				IF bMoveOnlyForwardAfterError THEN
					IF  (
						(ABS(LMOD(WheelAxisRef.NcToPlc.ActPos,360.0/nSlotsCount)) > (360.0/nSlotsCount*0.01)) AND
						(ABS(LMOD(WheelAxisRef.NcToPlc.ActPos,360.0/nSlotsCount)) < (360.0/nSlotsCount*0.99))  
						)
						AND NOT (LMOD(WheelAxisRef.NcToPlc.ActPos,360.0/nSlotsCount) = 0) 
					THEN                       
						 mcWheelMoveAbsolute.Position:=WheelAxisRef.NcToPlc.ActPos+360.0/nSlotsCount-LMOD(WheelAxisRef.NcToPlc.ActPos,360.0/nSlotsCount);
					ELSE
						mcWheelMoveAbsolute.Position:=WheelAxisRef.NcToPlc.ActPos;				
					END_IF 
				ELSE
					IF lrLastKnownPosition<>0 AND (ABS(ABS(lrLastKnownPosition)-ABS(WheelAxisRef.NcToPlc.ActPos))<(360.0/nSlotsCount*3)) THEN
						mcWheelMoveAbsolute.Position:=lrLastKnownPosition;
						mcWheelMoveAbsolute.Velocity:=lrVelocity;
						mcWheelMoveAbsolute.Acceleration:=lrAcceleration;
						mcWheelMoveAbsolute.Deceleration:=lrDeceleration;
						mcWheelPower.Override:=20;
						
						nTestW1:=nTestW1+1;
						(*Jak jest w ponad połowie ruchu to przesuwa się do przodu*) //Być może będzie trzeba przesuwać rejestr
						IF WheelAxisRef.NcToPlc.ActPos-lrLastKnownPosition > ((360.0/nSlotsCount)/2) THEN
							mcWheelMoveAbsolute.Position	:=	lrLastKnownPosition + 360.0/nSlotsCount;
							bMoveForward 					:=	TRUE; //Informacja że przesuneło się w prawo
							nTestW2 := nTestW2 + 1;
						END_IF
						
					ELSE
						IF LMOD(WheelAxisRef.NcToPlc.ActPos,360.0/nSlotsCount)>(360.0/nSlotsCount/2) THEN
							mcWheelMoveAbsolute.Position:=WheelAxisRef.NcToPlc.ActPos+360.0/nSlotsCount-LMOD(WheelAxisRef.NcToPlc.ActPos,360.0/nSlotsCount);
							nTestW3 := nTestW3 + 1;
						ELSE
							mcWheelMoveAbsolute.Position:=WheelAxisRef.NcToPlc.ActPos-LMOD(WheelAxisRef.NcToPlc.ActPos,360.0/nSlotsCount);
							nTestW4 := nTestW4 + 1;
						END_IF
						mcWheelMoveAbsolute.Velocity:=lrVelocity;
						mcWheelMoveAbsolute.Acceleration:=lrAcceleration;
						mcWheelMoveAbsolute.Deceleration:=lrDeceleration;
						mcWheelPower.Override:=20;
					END_IF
				END_IF*)
END_ACTION

END_FUNCTION_BLOCK

// ---- POUs/FB/F_StringToWstringPL.TcPOU
FUNCTION F_StringToWstringPL : WSTRING
VAR_INPUT
	sInput	: STRING;
END_VAR
VAR
	iNum			: INT;	
//	iChar			: INT;
	iLen			: INT;
END_VAR

iLen	:=LEN(sInput);	//ilość znaków w stringu
FOR iNum:=0 TO iLen-1 DO
	CASE sInput[iNum] OF
		
		140://Ś
			F_StringToWstringPL[iNum]	:= 90+256;
		143://Ź
			F_StringToWstringPL[iNum]	:= 121+256;	
		156://ś
			F_StringToWstringPL[iNum]	:= 91+256;
		159://ź
			F_StringToWstringPL[iNum]	:= 122+256;
		163://Ł
			F_StringToWstringPL[iNum]	:= 65+256;
		165://Ą
			F_StringToWstringPL[iNum]	:= 4+256;
		175://Ż
			F_StringToWstringPL[iNum]	:= 123+256;
		179://ł
			F_StringToWstringPL[iNum]	:= 66+256;
		185://ą
			F_StringToWstringPL[iNum]	:= 5+256;
		191://ż
			F_StringToWstringPL[iNum]	:= 124+256;
		198://Ć
			F_StringToWstringPL[iNum]	:= 6+256;
		202://Ę
			F_StringToWstringPL[iNum]	:= 24+256;	
		209://Ń
			F_StringToWstringPL[iNum]	:= 67+256;
//		211://Ó - bez zmiany
		230://ć
			F_StringToWstringPL[iNum]	:= 7+256;
		234://ę
			F_StringToWstringPL[iNum]	:= 25+256;
		241://ń
			F_StringToWstringPL[iNum]	:= 68+256;

//		243://ó - bez zmiany
		
		ELSE
			F_StringToWstringPL[iNum]	:= sInput[iNum];
	END_CASE

END_FOR
F_StringToWstringPL[iLen]:= 0;//Dodane 0 - koniec wstringa



//F_StringToWstringPL:="";

//FOR iNum:=1 TO LEN(sInput) DO
//	iChar	:= F_ToASC(MID(sInput,1,iNum));
//	CASE iChar OF
//		140:
//			F_StringToWstringPL	:= WCONCAT(F_StringToWstringPL,"Ś");
//		143:
//			F_StringToWstringPL	:= WCONCAT(F_StringToWstringPL,"Ź");
//		156:
//			F_StringToWstringPL	:= WCONCAT(F_StringToWstringPL,"ś");
//		159:
//			F_StringToWstringPL	:= WCONCAT(F_StringToWstringPL,"ź");
//		163:
//			F_StringToWstringPL	:= WCONCAT(F_StringToWstringPL,"Ł");
//		165:
//			F_StringToWstringPL	:= WCONCAT(F_StringToWstringPL,"Ą");
//		175:
//			F_StringToWstringPL	:= WCONCAT(F_StringToWstringPL,"Ż");	
//		179:
//			F_StringToWstringPL	:= WCONCAT(F_StringToWstringPL,"ł");
//		185:
//			F_StringToWstringPL	:= WCONCAT(F_StringToWstringPL,"ą");
//		191:
//			F_StringToWstringPL	:= WCONCAT(F_StringToWstringPL,"ż");
//		198:
//			F_StringToWstringPL	:= WCONCAT(F_StringToWstringPL,"Ć");
//		202:
//			F_StringToWstringPL	:= WCONCAT(F_StringToWstringPL,"Ę");		
//		209:
//			F_StringToWstringPL	:= WCONCAT(F_StringToWstringPL,"Ń");
//		211:
//			F_StringToWstringPL	:= WCONCAT(F_StringToWstringPL,"Ó");
//		230:
//			F_StringToWstringPL	:= WCONCAT(F_StringToWstringPL,"ć");
//		234:
//			F_StringToWstringPL	:= WCONCAT(F_StringToWstringPL,"ę");
//		241:
//			F_StringToWstringPL	:= WCONCAT(F_StringToWstringPL,"ń");
//		243:
//			F_StringToWstringPL	:= WCONCAT(F_StringToWstringPL,"ó");

		
//		ELSE
//			F_StringToWstringPL	:= WCONCAT(F_StringToWstringPL,TO_WSTRING(MID(sInput,1,iNum)));
			
//	END_CASE
//END_FOR

END_FUNCTION

// ---- POUs/P20_ExhaustFan.TcPOU
PROGRAM P20_ExhaustFan
VAR
	(*****************Wentylator wyciągaowy*******************)
	QbExhaustSystemEnable					AT %Q*	:BOOL;		
	IbExhaustSystemSwitchNormalMode			AT %I*	:BOOL;		
	IbExhaustSystemSwitchExMode				AT %I*	:BOOL;		
	IbExhaustSystemReady					AT %I*	:BOOL;		
	IbExhaustSystemAlarm					AT %I*	:BOOL;		
	IbExhaustSystemFlowOk					AT %I*	:BOOL;		
	IbExhaustSystemAlarmLevel1				AT %I*	:BOOL;		
			
	fbSensorAirFlow							: FB_SensorFlow;
	
END_VAR


QbExhaustSystemEnable := VIS.bExEnableShow OR bExEnable;

aSensors();

ExSensorWarning[1].sDescription:='Alarm poziomu 1 detekcja gazu 10%DGW';
IF (IbExhaustSystemAlarmLevel1 AND QbExhaustSystemEnable) AND NOT ExSensorWarning[1].bWarning THEN
	ExSensorWarning[1].bWarning		:=	TRUE;
ELSIF ( NOT IbExhaustSystemAlarmLevel1 )AND ExSensorWarning[1].bAcknowledge THEN
	ExSensorWarning[1].bWarning		:=	FALSE;
	ExSensorWarning[1].bAcknowledge	:=	FALSE;
	VIS.uliWarningAcknowledge.24 	:=	FALSE;
ELSIF ExSensorWarning[1].bAcknowledge THEN
	ExSensorWarning[1].bAcknowledge	:=	TRUE;
END_IF


ExhaustFanError;
IF ExhaustFanError.bReset THEN
	ExhaustFanError.bError				:= FALSE;
	ExhaustFanError.udiStationID		:= 0;
	ExhaustFanError.nErrorCode			:= 0;
	ExhaustFanError.bReset				:= FALSE;
	ExhaustFanError.sErrorString		:= '';
	ExhaustFanError.sErrorString2		:= '';	
END_IF
IF IbExhaustSystemAlarm AND QbExhaustSystemEnable AND NOT VIS.bErrorOccure THEN
	ExhaustFanError.bError				:= TRUE;
	ExhaustFanError.udiStationID		:= 75;
	ExhaustFanError.nErrorCode			:= 372;
	ExhaustFanError.bReset				:= FALSE;
	ExhaustFanError.sErrorString		:= 'System wentylacji Ex - błąd - sprawdź szafę R4 Ex';
	ExhaustFanError.sErrorString2		:= '';
ELSIF NOT QbExhaustSystemEnable THEN
	ExhaustFanError.bError				:= FALSE;
END_IF

ACTION aSensors:
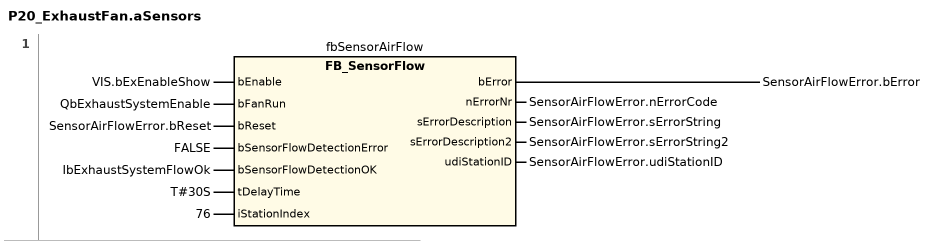
// NETWORK 1
fbSensorAirFlow(
    bEnable := VIS.bExEnableShow,
    bFanRun := QbExhaustSystemEnable,
    bReset := SensorAirFlowError.bReset,
    bSensorFlowDetectionError := FALSE,
    bSensorFlowDetectionOK := IbExhaustSystemFlowOk,
    tDelayTime := T#30S,
    iStationIndex := 76,
    nErrorNr => SensorAirFlowError.nErrorCode,
    sErrorDescription => SensorAirFlowError.sErrorString,
    sErrorDescription2 => SensorAirFlowError.sErrorString2,
    udiStationID => SensorAirFlowError.udiStationID); // FB_SensorFlow
SensorAirFlowError.bError := fbSensorAirFlow.bError;
END_ACTION

END_PROGRAM

// ---- POUs/FB/NewFBs/FB_SensorFlow.TcPOU
FUNCTION_BLOCK FB_SensorFlow
VAR_INPUT
	bEnable										:	BOOL;
	bFanRun										: 	BOOL;
	bReset										:	BOOL;
	bSensorFlowDetectionError				 	:	BOOL;			//Czujnik detekcji przeblywy bląd
	bSensorFlowDetectionOK					 	:	BOOL;			// Nie ma przeblywy
	tDelayTime									:	TIME;
	iStationIndex								:	UDINT;
END_VAR
	
VAR_OUTPUT
	bError										:	BOOL;
	nErrorNr									: 	UDINT;							//Nr błędu grzałki zasadniczej
	sErrorDescription							: 	STRING(200);	
	sErrorDescription2							: 	STRING(200);	
	udiStationID								:	UDINT;				// Nr stacji	
END_VAR
VAR
	tonSensorDelay								:	TON;
END_VAR

ACT_Cycle();
aStationID();

ACTION ACT_Cycle:
tonSensorDelay(IN:=(bEnable AND NOT bSensorFlowDetectionOK AND bFanRun),PT:=tDelayTime);

IF (NOT bError) THEN
	
	IF (bSensorFlowDetectionError) THEN
		bError 							:= FALSE;
		sErrorDescription 				:= 'Błąd czujnika przepływy';
		sErrorDescription2 				:= '';
		nErrorNr						:= 363;
	END_IF
	
	IF (tonSensorDelay.Q AND NOT bError) THEN
		bError 							:= FALSE;
		sErrorDescription 				:= 'Nie ma potwierdzenie przepływy od czujnika';
		sErrorDescription2 				:= '';
		nErrorNr						:= 364;
	END_IF
END_IF

IF (bReset) THEN
	bError 							:= FALSE;
	sErrorDescription 				:= '';
	sErrorDescription2 				:= '';
	nErrorNr						:= 0;
END_IF
END_ACTION

ACTION aStationID:
udiStationID	:=	iStationIndex;
END_ACTION

END_FUNCTION_BLOCK

// ---- POUs/P06_LidPuttedCheck.TcPOU
{attribute 'TcContextName' := 'PlcTask'}
PROGRAM P06_LidPuttedCheck
VAR
	fbLidPuttedCheck										: FB_VisionChecker;
	eLidPuttedCheckState									: E_Station; 			// Stan pracy podajnika platynek			
	eLidPuttedCheckRunningState								: E_CheckerState; 		// Stan pracy podajnika platynek
	fbLidPuttedCheckState									: FB_State;
	
	IbLidPuttedCheckHeightEncoderPulses 			AT %I*	: BOOL;	
	QbLidPuttedCheckHeightUpCmd 					AT %Q*	: BOOL; 				// Wyjście sterujące podnośnikiem sprawdzania platynki, Silnik w górę
	QbLidPuttedCheckHeightDownCmd 					AT %Q*	: BOOL; 				// Wyjście sterujące podnośnikiem sprawdzania platynki, Silnik w dół
	
	//Kamera do sprawdzania platynek
	IbLidPuttedCheckCameraError						AT %I*	: BOOL; 						
	IbLidPuttedCheckCameraGood						AT %I*	: BOOL; 						 
	IbLidPuttedCheckCameraBusy						AT %I*	: BOOL; 
	IuiLidPuttedCheckCameraProgram					AT %I*	: UINT; 
	
	QbLidPuttedCheckCameraTrigger					AT %Q*	: BOOL; 						
	QuiLidPuttedCheckCameraProgram					AT %Q*	: UINT; 
	QbLidPuttedCheckCameraChangeProgram				AT %Q*	: BOOL; 	
	
	TimerLidPuttedCheckEnable								: TOF;
	rtEnable												: R_TRIG;
	bTemp													: BOOL;

	IbLidPuttedCheck11Sensor						AT %I*	: BOOL; 	
	IbLidPuttedCheck12Sensor						AT %I*	: BOOL; 	
	IbLidPuttedCheck13Sensor						AT %I*	: BOOL; 	
	IbLidPuttedCheck21Sensor						AT %I*	: BOOL; 	
	IbLidPuttedCheck22Sensor						AT %I*	: BOOL; 	
	IbLidPuttedCheck23Sensor						AT %I*	: BOOL; 		
	
END_VAR

ACT_LidPuttedCheck();

(* BAZOWANIE - ZMIAN*)
rtEnable(CLK := fbLidPuttedCheck.bEnable, Q =>);
IF rtEnable.Q AND (P00_PackML.fbPMLAuto.ePMLState = Tc3_PackML.E_PMLState.ePMLState_IDLE OR 
   P00_PackML.fbPMLAuto.ePMLState = Tc3_PackML.E_PMLState.ePMLState_EXECUTE) THEN
   
   // VIS.bLidPuttedCheckHeightSet := TRUE;
	
ELSIF fbLidPuttedCheck.eState = E_Station.eHomingDone OR VIS.bErrorOccure THEN
	
   // VIS.bLidPuttedCheckHeightSet := FALSE;
	
END_IF
(*KONIEC BAZOWANIE - ZMIANA*)

(********* GENEROWANIE STANU STACJI DO WIZKI**********)
fbLidPuttedCheckState(
	eState					:= eLidPuttedCheckState , 
	bRun					:= P00_PackML.fbPMLAuto.ePMLState = Tc3_PackML.E_PMLState.ePMLState_EXECUTE,	
	eCheckerRunningState	:= eLidPuttedCheckRunningState , 
	sStateDesc				=> VIS.sLidPuttedCheckState,
	iState					=> VIS.iLidPuttedCheckState );
(***** KONIEC GENEROWANIE STANU STACJI DO WIZKI*******)	

(*Opoznienie wyłączanie enabla*)
TimerLidPuttedCheckEnable (IN := bLidPuttedCheckEnable , PT:=T#2S);

ACTION ACT_LidPuttedCheck:
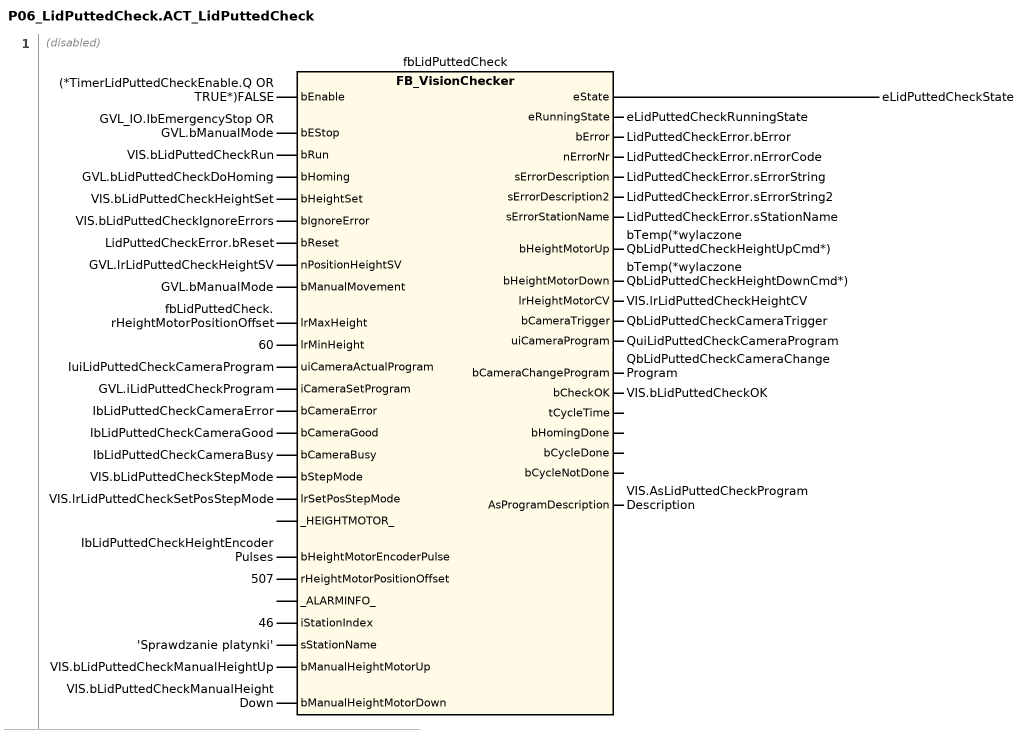
// NETWORK 1 (disabled)
// fbLidPuttedCheck(
//     bEnable := (*TimerLidPuttedCheckEnable.Q OR TRUE*)FALSE,
//     bEStop := GVL_IO.IbEmergencyStop OR GVL.bManualMode,
//     bRun := VIS.bLidPuttedCheckRun,
//     bHoming := GVL.bLidPuttedCheckDoHoming,
//     bHeightSet := VIS.bLidPuttedCheckHeightSet,
//     bIgnoreError := VIS.bLidPuttedCheckIgnoreErrors,
//     bReset := LidPuttedCheckError.bReset,
//     nPositionHeightSV := GVL.lrLidPuttedCheckHeightSV,
//     bManualMovement := GVL.bManualMode,
//     lrMaxHeight := fbLidPuttedCheck.rHeightMotorPositionOffset,
//     lrMinHeight := 60,
//     uiCameraActualProgram := IuiLidPuttedCheckCameraProgram,
//     iCameraSetProgram := GVL.iLidPuttedCheckProgram,
//     bCameraError := IbLidPuttedCheckCameraError,
//     bCameraGood := IbLidPuttedCheckCameraGood,
//     bCameraBusy := IbLidPuttedCheckCameraBusy,
//     bStepMode := VIS.bLidPuttedCheckStepMode,
//     lrSetPosStepMode := VIS.lrLidPuttedCheckSetPosStepMode,
//     bHeightMotorEncoderPulse := IbLidPuttedCheckHeightEncoderPulses,
//     rHeightMotorPositionOffset := 507,
//     iStationIndex := 46,
//     sStationName := 'Sprawdzanie platynki',
//     bManualHeightMotorUp := VIS.bLidPuttedCheckManualHeightUp,
//     bManualHeightMotorDown := VIS.bLidPuttedCheckManualHeightDown,
//     eRunningState => eLidPuttedCheckRunningState,
//     bError => LidPuttedCheckError.bError,
//     nErrorNr => LidPuttedCheckError.nErrorCode,
//     sErrorDescription => LidPuttedCheckError.sErrorString,
//     sErrorDescription2 => LidPuttedCheckError.sErrorString2,
//     sErrorStationName => LidPuttedCheckError.sStationName,
//     bHeightMotorUp => bTemp(*wylaczone QbLidPuttedCheckHeightUpCmd*),
//     bHeightMotorDown => bTemp(*wylaczone QbLidPuttedCheckHeightDownCmd*),
//     lrHeightMotorCV => VIS.lrLidPuttedCheckHeightCV,
//     bCameraTrigger => QbLidPuttedCheckCameraTrigger,
//     uiCameraProgram => QuiLidPuttedCheckCameraProgram,
//     bCameraChangeProgram => QbLidPuttedCheckCameraChangeProgram,
//     bCheckOK => VIS.bLidPuttedCheckOK,
//     AsProgramDescription => VIS.AsLidPuttedCheckProgramDescription); // FB_VisionChecker
// eLidPuttedCheckState := fbLidPuttedCheck.eState;
END_ACTION

END_PROGRAM

// ---- POUs/FB/FB_VisionChecker.TcPOU
(*
Nazwa:			FB_VisionChecker
Opis:			stacja sprawdzania platynek czujnikiem wizyjnym
Wersja:			v1.0
Data:			2023-05-30
Autor:			DP
Urzadzenia:		Czujnik wizyjny KEYENCE
Konfiguracja:	
Info:
- 
*)

FUNCTION_BLOCK FB_VisionChecker
VAR_INPUT
	bEnable:BOOL;				//Zezowlenie na pracę stacji sprawdzania
	bEStop:BOOL;				//Stop Awaryjny nieaktywny
	bRun:BOOL;					//Rozkaz łapania 	
	bHoming:BOOL;				//Zezwolenie na wykonanie bazowania i pozycjonowania stacji sprawdzania
	bHeightSet:BOOL;			//Ustaw wysokość
	bIgnoreError:BOOL;			//Ignorowania błędów cyklu pracy
	bReset:BOOL;				//Reset błędu, jeśli w stanie "eError"
	nPositionHeightSV:LREAL;	//Wysokość zadana na której ma znajdować się stacja sprawdzania
	bManualMovement:BOOL; 		//Uruchomienie trybu ruchów ręcznych
	lrMaxHeight:LREAL;			//Maksymalna wysokość stacji sprawdzania
	lrMinHeight:LREAL;			//Minimalna wysokość stacji sprawdzania
	uiCameraActualProgram:UINT;
	iCameraSetProgram:INT;
	bCameraError:BOOL; 
	bCameraGood:BOOL; 	
	bCameraBusy:BOOL; 	
	//StepMode
	bStepMode				: BOOL;		//Włączony tryb skokowy sterowania podnośnikami (tylko w serwisie)
	lrSetPosStepMode		: LREAL; 	//Ruch podnośnika o zadaną wartość w trybie krokowym (tylko w serwisie)
	
	_HEIGHTMOTOR_ :BOOL;	
	bHeightMotorEncoderPulse :BOOL;			//Sygnał impulsów enkodera siłownika
	rHeightMotorPositionOffset :REAL;		//Wysokość bazowani podnośnika

	_ALARMINFO_ :BOOL;
	iStationIndex:UDINT;					//Numer stacji 
	sStationName:STRING;					//Nazwa stacji	

END_VAR
VAR_OUTPUT	
	eState: E_Station;						//Stan ogólny bloku
	eRunningState: E_CheckerState;			//Stan stacji sprawdzania
	bError: BOOL;							//Błąd stacji
	nErrorNr: UDINT;						//Nr błędu stacji sprawdzania
	sErrorDescription:STRING(200);			//Opis błędu
	sErrorDescription2:STRING(200);			//Opis błędu
	sErrorStationName:STRING;				//Nazwa stacji
	bHeightMotorUp:BOOL;					//Sterowanie silnikiem podnośnika  - RUCH W GÓRĘ
	bHeightMotorDown:BOOL;					//Sterowanie silnikiem podnośnika  - RUCH W DÓŁ
	lrHeightMotorCV:LREAL;					//Aktualna wysokość stacji sprawdzania
	bCameraTrigger:BOOL; 
	uiCameraProgram:UINT; 
	bCameraChangeProgram:BOOL; 	
	bCheckOK:BOOL;							//Platynka OK
	tCycleTime:TIME;	
	bHomingDone:BOOL;						//Wymagane ponowne bazowanie (blad podczas bazowania lub stop awaryjny)
	bCycleDone:BOOL;
	bCycleNotDone:BOOL;
	AsProgramDescription: ARRAY [0..20] OF STRING;	// Opis programów

END_VAR
VAR
	tonHeightNoChange: TON; // Timer wykrycia braku ruchu siłownika zmiany wysokości stacji
	nLastPositionHeightCV: LREAL;// Pozycja podnośnika w poprzednim cyklu programu
	tonErrorHeightChange: TON; // Timer błędu podnośnika
	rtEncoderHomed:R_TRIG;
	tonCycleTimer:TON;
	rtrigCycleTimerRead:R_TRIG;
	tonTriggerDelay: TON;
	tonNotBusyDelay: TON;
	tonLidNOK: TON;
	tofMotorUpPermition: TOF;
	tofMotorDownPermition: TOF;
	tonLimitPosMinReachedDelay: TON;
	tonLimitPosMaxReachedDelay: TON;
	tonMaxHeight: TON;
	tonMinHeight: TON;
	
	//Podnośnik Jiesang	
	fbHeightMotorEncoder: FB_JiesangActuatorEncoder_1;	// Blok enkodera podnośnika chwytaka stabilizującego pod zakręcarką	
	bHeightMotorEncoderCounterReset:BOOL; 				// Sygnał resetu enkodera
	bHeightMotorEncoderHomed:BOOL;						// Informacja od enkodera że jest zbazowany

	eLastState: E_Station;								// Stan ogólny bloku
	eLastRunningState: E_CheckerState;					// Stan podbloku
	eLastStateTemp: E_Station;							// Stan ogólny bloku
	eLastRunningStateTemp: E_CheckerState;				// Stan podbloku	
	
	bStateError: BOOL;

	//Step Mode
	rtStepModeUp			: R_TRIG;
	rtStepModeDown			: R_TRIG;
	lrStepModeHeightMotorSV	: LREAL;
	bStepModeMoving			: BOOL;
	tofStepModeMoving		: TOF;	
	rtCheckingEnd			: R_TRIG;
	tonbCameraChangeProgram: TON;
	rtuiCameraActualProgram: R_TRIG;
	tonTryChangeProgram: TON;
	
	//Zmienne od EVENTLOGGER
	bAlarmInit 						: BOOL := TRUE; 
	nAlarmNumerator					: INT;
	arfbAlarm						: ARRAY[0..19] OF  FB_TcAlarm;		//Tablica bloczków błędów
	fbSourceInfo 					: FB_TcSourceInfo;
	iSourceInfo						: I_TcSourceInfo;
	sAlarmTest						: STRING;
	//Koniec zmiennych od EVENTLOGGER
END_VAR

VAR_IN_OUT
	bManualHeightMotorUp:BOOL;			//Ruch ręczny podnośnika stacji w górę
	bManualHeightMotorDown:BOOL;		//Ruch ręczny podnośnika stacji w dół
END_VAR

HeightMotor();
ErrorHandling();
Control();
Statistics();
Programs();

(*Zapisywanie ostatniego stanu*)
IF eLastStateTemp<>eState THEN
	eLastState := eLastStateTemp;
END_IF
eLastStateTemp := eState;
IF eLastRunningStateTemp<>eRunningState THEN
	eLastRunningState := eLastRunningStateTemp;
END_IF
eLastRunningStateTemp := eRunningState;
(*Koniec Zapisywanie ostatniego stanu*)

nLastPositionHeightCV:=lrHeightMotorCV;

ACTION Control:

	(** TIMERY**)
	rtEncoderHomed				(CLK:=bHeightMotorEncoderHomed,																Q=>);
	tonHeightNoChange			(IN:=((bHeightMotorUp OR bHeightMotorDown) AND (nLastPositionHeightCV=lrHeightMotorCV)), 	PT:=T#1S); 
	tonLimitPosMinReachedDelay	(IN:=(lrHeightMotorCV<=lrMinHeight) AND eState=E_Station.eHoming,							PT:=T#2S);
	tonLimitPosMaxReachedDelay	(IN:=(lrHeightMotorCV>=lrMaxHeight) AND eState=E_Station.eHoming,							PT:=T#2S);

	(*****Wyłączenie enable*****)
	IF NOT bEnable THEN
		IF eState <> E_Station.eDisabled AND eState <> E_Station.ePreparingToDisable THEN
				eState 							:=	E_Station.ePreparingToDisable; 
		END_IF	
	END_IF

	(*****Estop*****)
	IF NOT bEstop  THEN	
		IF eState <> E_Station.eAborted AND eState <> E_Station.eAborting AND eState <> E_Station.eDisabled THEN
				eState 							:=	E_Station.eAborting; 
		END_IF
	END_IF

	
	CASE eState OF
	/////////////////////////////	
		E_Station.eDisabled: 					// Stan nieaktywnosci (Stacja wyłączona) 
		
			IF bEnable THEN
				eState 							:=	E_Station.ePreparingToReady; 
			END_IF 
			
    /////////////////////////////	    
		E_Station.eAborted: 					// Stan bezpiecznego zatrzymania (po Abortingu) 

			IF bEStop THEN
				eState 							:=	E_Station.ePreparingToReady;
			END_IF
			
	/////////////////////////////	
		E_Station.eAborting:                 	// Stan bezpiecznego zatrzymywania (po EStopie)
			
			bHeightMotorUp						:=	FALSE;
			bHeightMotorDown					:=	FALSE;
			eState 								:=	E_Station.eAborted;  
			eRunningState						:=	E_CheckerState.eDisabled;
			
	/////////////////////////////			
		E_Station.eError:                 	 	// Stan błędu 	
	
			IF bReset THEN
				eState 							:=	E_Station.eResetting;
			ELSE
				ResetCommands();
			END_IF
			
	/////////////////////////////
		E_Station.eResetting:					// Stan resetowania bledu (po Errorze)
			
			bError := FALSE;
			IF NOT bError THEN
				nErrorNr 						:=	0;
   				sErrorDescription 				:=	'';
				eState 							:=	E_Station.ePreparingToReady;
			ELSE
				eState 							:=	E_Station.eError;
			END_IF
        
	/////////////////////////////
		E_Station.eManualMovement:     			// Stan ruchów manualnych  
       
			ManualMovements();
			//Wyjście z trybu serwisowego
			IF NOT bManualMovement THEN
				bHeightMotorUp					:=	FALSE;
				bHeightMotorDown				:=	FALSE;	
				eState							:=	E_Station.eReady;
			END_IF

	/////////////////////////////
		E_Station.eHoming:						// Stan bazowania 

			Homing();
			IF NOT bHoming AND NOT bHeightSet THEN
				bHeightMotorDown				:=	FALSE;
				bHeightMotorUp					:=	FALSE;
				eState							:=	E_Station.ePreparingToReady;
			END_IF		
			
	/////////////////////////////
		E_Station.eHomingDone:                  // Stan wykonania bazowania 
		
			bHeightMotorDown					:=	FALSE;
			bHeightMotorUp						:=	FALSE;
			bHeightMotorEncoderCounterReset		:=	FALSE;
			bHomingDone							:=	TRUE;
			IF NOT bHoming AND NOT bHeightSet THEN
			   eState							:=	E_Station.eReady;
			END_IF
			
	/////////////////////////////
		E_Station.ePreparingToReady:            // Stan przygotowywania do gotowosci (zawsze przed Ready)  
		
			eRunningState						:=	E_CheckerState.eReady;
			eState								:=	E_Station.eReady;	
			
	/////////////////////////////
		E_Station.ePreparingToDisable:          // Stan przygotowywania do nieaktywnosci (po wyłączeniu Enable) 
  
			bHeightMotorUp						:=	TRUE;
			bHeightMotorDown					:=	FALSE;	
			IF tonHeightNoChange.Q THEN
				bHeightMotorUp					:=	FALSE;
				eState							:=	E_Station.eDisabled;
				eRunningState					:=	E_CheckerState.eDisabled;
			END_IF	
				
	/////////////////////////////
		E_Station.eReady:						// Stan gotowosci 
			
			IF bRun AND NOT bCycleDone AND NOT bCycleNotDone THEN
				eState 							:=	E_Station.eStarting; 
			END_IF
			IF bHoming OR bHeightSet THEN
				eState 							:=	E_Station.eHoming; 
			END_IF
			IF bManualMovement THEN
				//Jeśli przejście w tryb ruchów manualnych przepisz wszystkie stany siłowników sterowanych przez moduł
				//aby zapobiec ewentualnym kolizjom po wejściu w tryb serwisowy
				bManualHeightMotorUp			:=	bHeightMotorUp;
				bManualHeightMotorDown			:=	bHeightMotorDown;
				eState 							:=	E_Station.eManualMovement; 
			END_IF
			IF NOT bRun THEN
				bCycleDone 						:=	FALSE;
				bCycleNotDone 					:=	FALSE;			
			END_IF
			
	/////////////////////////////
		E_Station.eStopping:					// Stan zatrzymywania 
			
			Running();
			bCameraTrigger						:= FALSE;
			bCheckOK							:= FALSE;
			eState								:=	E_Station.eReady;
			
	/////////////////////////////
		E_Station.eStarting:                  	// Stan uruchamiania (po Ready)
		
			eRunningState						:= E_CheckerState.eReady;
			eState								:= E_Station.eRunning; 

	/////////////////////////////
		E_Station.eRunning:               		// Stan wykonywania cyklu (po Startingu), w tym stanie osobny
 
			Running();
			IF NOT bRun THEN 					(*Przerywanie cyklu*)
				eState							:=	E_Station.eStopping;
				bCycleNotDone					:=	TRUE;
			END_IF
			(*IF bCycleDone OR bCycleNotDone THEN (*Cykl zakończony*)
				eState 				 := E_Station.eReady;
			END_IF*)						
			
	/////////////////////////////		
	END_CASE
END_ACTION

ACTION ErrorHandling:
// Alarm_0360	360	Error	Blokada podnośnika lub brak zasilania - sprawdź czujnik lub odblokuj mechanicznie
// Alarm_0361	361	Error	Wartość zadana wysokości jest większa od maksymalnej - zmień ustawienia w recepturze
// Alarm_0362	362	Error	Wartość zadana wysokości jest mniejsza od minimalnej - zmień ustawienia w recepturze

IF bAlarmInit THEN
    bAlarmInit := FALSE; 
	fbSourceInfo.Clear();
	fbSourceInfo.sName:=sStationName;//'Machine';
	fbSourceInfo.nId:=iStationIndex;//2700;
	// Alarm_0360	360	Error	Blokada podnośnika lub brak zasilania - sprawdź czujnik lub odblokuj mechanicznie
    arfbAlarm[0].CreateEx(stEventEntry := TC_EVENTS.AlarmClass.Alarm_0360, bWithConfirmation:= FALSE,  ipSourceInfo:= fbSourceInfo); 
	// Alarm_0361	361	Error	Wartość zadana wysokości jest większa od maksymalnej - zmień ustawienia w recepturze
	arfbAlarm[1].CreateEx(stEventEntry := TC_EVENTS.AlarmClass.Alarm_0361, bWithConfirmation:= FALSE,  ipSourceInfo:= fbSourceInfo);
	// Alarm_0362	362	Error	Wartość zadana wysokości jest mniejsza od minimalnej - zmień ustawienia w recepturze
	arfbAlarm[2].CreateEx(stEventEntry := TC_EVENTS.AlarmClass.Alarm_0362, bWithConfirmation:= FALSE,  ipSourceInfo:= fbSourceInfo);
END_IF

//OBSŁUGA BŁĘDÓW STACJI SPRAWDZANIA

//************LISTA BŁĘDÓW***************
bStateError:= (eState=E_Station.eError) OR (eState=E_Station.eResetting) OR bIgnoreError;

IF bEnable THEN
	// Alarm_0360	360	Error	Blokada podnośnika lub brak zasilania - sprawdź czujnik lub odblokuj mechanicznie
	//Error 1 - podnośnik nie porusza się pomimo wysterowania 
	tonErrorHeightChange(IN:=(bHeightMotorUp OR bHeightMotorDown) AND nLastPositionHeightCV=lrHeightMotorCV, PT:=T#3S);
	IF tonErrorHeightChange.Q THEN
		IF NOT arfbAlarm[0].bActive THEN
			bHeightMotorUp:=FALSE;
			bHeightMotorDown:=FALSE;
			arfbAlarm[0].Raise(nTimeStamp:=0);
		END_IF
	ELSE	
		IF  arfbAlarm[0].bActive AND bReset THEN
			arfbAlarm[0].Clear(nTimeStamp:=0, bResetConfirmation:= FALSE);
		END_IF	
// 		bHeightMotorUp:=FALSE;
// 		bHeightMotorDown:=FALSE;
// 		bError := TRUE;
// 		nErrorNr:=241;
// 		//nErrorNr := nErrorNr+iStationIndex;
// 		sErrorDescription:='Blokada podnośnika lub brak zasilania - sprawdź czujnik lub odblokuj mechanicznie';	
	END_IF
	// Alarm_0361	361	Error	Wartość zadana wysokości jest większa od maksymalnej - zmień ustawienia w recepturze
	//Error 7 - Bład nastaw max
	tonMaxHeight(IN:=nPositionHeightSV>lrMaxHeight AND NOT bHomingDone AND eState=E_Station.eStarting,PT:=T#0S);
	IF tonMaxHeight.Q THEN
		arfbAlarm[1].ipArguments.Clear() .AddLReal(lrMaxHeight);
		IF NOT arfbAlarm[1].bActive THEN
			bHeightMotorUp:=FALSE;
			bHeightMotorDown:=FALSE;
			arfbAlarm[1].Raise(nTimeStamp:=0);
		END_IF
	ELSE	
		IF  arfbAlarm[1].bActive AND bReset THEN
			arfbAlarm[1].Clear(nTimeStamp:=0, bResetConfirmation:= FALSE);
		END_IF	
// 		bHeightMotorUp:=FALSE;
// 		bHeightMotorDown:=FALSE;
// 		bError := TRUE;
// 		nErrorNr:=242;
// 		//nErrorNr := nErrorNr+iStationIndex;
// 		sErrorDescription:='Wartość zadana wysokości jest większa od maksymalnej - zmień ustawienia w recepturze';
// 		sErrorDescription2:=REAL_TO_STRING(LREAL_TO_INT(lrMaxHeight));
	END_IF
	// Alarm_0362	362	Error	Wartość zadana wysokości jest mniejsza od minimalnej - zmień ustawienia w recepturze
	//Error 8 - Bład nastaw min
	//tonMinHeight(IN:=nPositionHeightSV<lrMinHeight AND NOT bHomingDone AND eState=E_Station.eStarting,PT:=T#0S);
	//IF tonMinHeight.Q AND NOT bStateError THEN
	//	bHeightMotorUp:=FALSE;
	//	bHeightMotorDown:=FALSE;
	//	bError := TRUE;
	//	nErrorNr:=243;
	//	//nErrorNr := nErrorNr+iStationIndex;
	//	sErrorDescription:='Wartość zadana wysokości jest mniejsza od minimalnej - zmień ustawienia w recepturze';
	//	sErrorDescription2:=REAL_TO_STRING(LREAL_TO_INT(lrMinHeight));	
	//END_IF

ELSE
	bError := FALSE;
END_IF

	
//******************PRZEJŚCIE DO eERROR*****************************

IF bError AND NOT bStateError THEN
	IF eLastState = eRunning THEN
		bCycleNotDone := TRUE;
	END_IF
	eState := E_Station.eError;
END_IF

//****************WYŚWIETLANIE STATUSU BLEDU***********************

(*Wyświetlanie błedu na wyjściu*)
bError							:= FALSE;
FOR nAlarmNumerator := 0 TO 19 DO
	bError						:= bError OR arfbAlarm[nAlarmNumerator].bActive;
END_FOR

(*Przepisywanie nazwy stacji*)
sErrorStationName := sStationName;

//Jezeli nie zbazowane to potrzebne bazowanie
IF NOT bHeightMotorEncoderHomed  THEN
	bHomingDone:=FALSE;
END_IF
END_ACTION

ACTION HeightMotor:
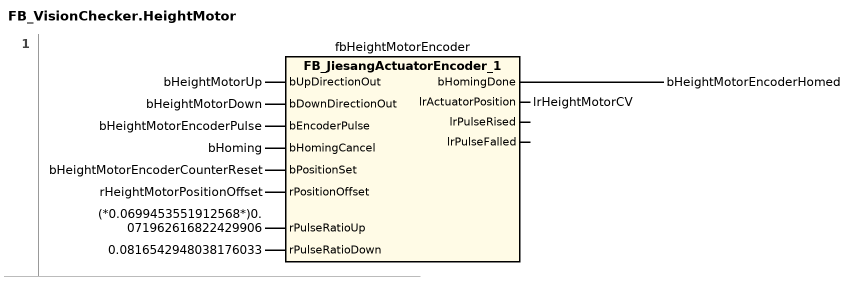
// NETWORK 1
fbHeightMotorEncoder(
    bUpDirectionOut := bHeightMotorUp,
    bDownDirectionOut := bHeightMotorDown,
    bEncoderPulse := bHeightMotorEncoderPulse,
    bHomingCancel := bHoming,
    bPositionSet := bHeightMotorEncoderCounterReset,
    rPositionOffset := rHeightMotorPositionOffset,
    rPulseRatioUp := (*0.0699453551912568*)0.071962616822429906,
    rPulseRatioDown := 0.0816542948038176033,
    lrActuatorPosition => lrHeightMotorCV); // FB_JiesangActuatorEncoder_1
bHeightMotorEncoderHomed := fbHeightMotorEncoder.bHomingDone;
END_ACTION

ACTION Homing:
//BAZOWANIE

	
//Podnoszenie stacji do maksymalnej pozycji
IF NOT bHeightMotorEncoderHomed OR rtEncoderHomed.Q THEN
	bHeightMotorUp:=TRUE;
	bHeightMotorDown:=FALSE;
	IF tonHeightNoChange.Q THEN
		bHeightMotorEncoderCounterReset:=TRUE;
		bHeightMotorUp:=FALSE;
    END_IF
	//Jesli enkoder zbazowany zakończ bazowanie	
	IF rtEncoderHomed.Q THEN
		bHeightMotorUp:=FALSE;
		bHeightMotorDown:=FALSE;
		eState:=E_Station.eHomingDone;
	END_IF		
		
//Po podniesieniu stacji opuszczanie do ustalonej wysokości
ELSIF bHeightMotorEncoderHomed THEN
	bHeightMotorEncoderCounterReset:=FALSE;
	bHeightMotorUp:=lrHeightMotorCV<=nPositionHeightSV;
	bHeightMotorDown:=lrHeightMotorCV>=nPositionHeightSV;
	//Kiedy stacja osiągnie wysokość zadaną
	IF ABS(lrHeightMotorCV-nPositionHeightSV)<1 OR tonLimitPosMaxReachedDelay.Q OR tonLimitPosMinReachedDelay.Q THEN
		bHeightMotorDown:=FALSE;
		bHeightMotorUp:=FALSE;
		eState:=E_Station.eHomingDone;
	END_IF			
END_IF
END_ACTION

ACTION ManualMovements:

//W trybie ruchów manualnych wykonuj ruchy za pomocą rozkazów manualnych
IF NOT bRun THEN
	eRunningState		:=	E_CheckerState.eReady;
	bCameraTrigger		:=	FALSE;
	bCheckOK			:=	FALSE;
	bHeightMotorUp		:=	bManualHeightMotorUp;
	bHeightMotorDown	:=	bManualHeightMotorDown;
ELSE	//Kasuje zeby po cyklu nic sie nie poruszało
	bManualHeightMotorUp  := FALSE;
	bManualHeightMotorDown  := FALSE;
END_IF


IF bHoming OR bHeightSet THEN
	eState:=E_Station.eHoming;
END_IF
	
Running();
ManualMovementsStepMode();
	
//Zabezpieczenie przed kolizją stacji poprzez ruch podnośnika	
IF bHeightMotorDown AND lrHeightMotorCV<=lrMinHeight AND NOT bHoming AND NOT bHeightSet THEN
	bHeightMotorDown:=FALSE;
END_IF	

IF bHeightMotorUp AND lrHeightMotorCV>=lrMaxHeight AND NOT bHoming AND NOT bHeightSet THEN
	bHeightMotorUp:=FALSE;
END_IF
END_ACTION

ACTION ManualMovementsStepMode:
bManualHeightMotorUp;
bManualHeightMotorDown;
bStepMode;		
lrSetPosStepMode;

// Limity
IF lrSetPosStepMode < 1			THEN	lrSetPosStepMode := 1;	END_IF
IF lrSetPosStepMode > 10		THEN	lrSetPosStepMode := 10;	END_IF

// Zabezpieczenie przed zbyt szybkim włączaniem
tofStepModeMoving				(IN := bStepModeMoving,					PT:=T#500MS);

// Możliwe włączenie jeżeli zakończyło poprzedni ruch
rtStepModeUp					(CLK :=	bStepMode AND NOT tofStepModeMoving.Q	AND bManualHeightMotorUp,	Q=>);
rtStepModeDown					(CLK :=	bStepMode AND NOT tofStepModeMoving.Q 	AND bManualHeightMotorDown,	Q=>);

// Włączenie ruchu w górę
IF rtStepModeUp.Q THEN
	bStepModeMoving				:= TRUE;
	bManualHeightMotorUp		:= FALSE;
	bManualHeightMotorDown		:= FALSE;
	lrStepModeHeightMotorSV		:= lrHeightMotorCV	+	lrSetPosStepMode;
END_IF

// Włączenie ruchu w dół
IF rtStepModeDown.Q THEN
	bStepModeMoving				:= TRUE;
	bManualHeightMotorUp		:= FALSE;
	bManualHeightMotorDown		:= FALSE;
	lrStepModeHeightMotorSV		:= lrHeightMotorCV	-	lrSetPosStepMode;
END_IF
// DODAĆ RESET bStepModeMoving PO BLEDZIE!
// Ruch w górę !SPRAWDZIC ZNAKI!
IF bStepModeMoving THEN
	bHeightMotorUp				:=	lrHeightMotorCV	<=	lrStepModeHeightMotorSV;
	bHeightMotorDown			:=	lrHeightMotorCV	>=	lrStepModeHeightMotorSV;	
	
	IF ABS(lrHeightMotorCV-lrStepModeHeightMotorSV) < 0.5	OR	// Pozycja osiągnięta (co do 1mm)
			(lrHeightMotorCV<=lrMinHeight)				OR 	// Pozycja poniżej minimalnej
			(lrHeightMotorCV>=lrMaxHeight) 					// Pozycja powyżej maksymalnej
	THEN
		bHeightMotorDown		:= FALSE;
		bHeightMotorUp			:= FALSE;
		bStepModeMoving			:= FALSE;
	END_IF	
END_IF
END_ACTION

ACTION Programs:
tonbCameraChangeProgram	(IN:=bCameraChangeProgram,PT:=T#1S);
tonTryChangeProgram	(IN:=uiCameraActualProgram <> uiCameraProgram AND NOT bCameraChangeProgram, PT:=T#5S);
rtuiCameraActualProgram	(CLK:=uiCameraActualProgram <> uiCameraProgram,	Q=>);
uiCameraProgram	:=	INT_TO_UINT(iCameraSetProgram);

IF rtuiCameraActualProgram.Q	 OR  tonTryChangeProgram.Q THEN
	bCameraChangeProgram	:=	TRUE;
END_IF
IF tonbCameraChangeProgram.Q THEN
	bCameraChangeProgram	:=	FALSE;
END_IF

(*Narzędzia*)
AsProgramDescription[0] := '1. opak:225082(elite), platynka:241081(~55mm)';
AsProgramDescription[1] := '2. opak:220505(wega), platynka:soraya 240964(54mm)';
AsProgramDescription[2] := '3. opak:220395(shine), platynka:bielenda 241181(57mm)';
AsProgramDescription[3] := '4. opak:rezerwa, platynka:rezerwa';
AsProgramDescription[4] := '5. opak:rezerwa, platynka:rezerwa';
AsProgramDescription[5] := '6. opak:rezerwa, platynka:rezerwa';
AsProgramDescription[6] := '7. opak:rezerwa, platynka:rezerwa';
AsProgramDescription[7] := '8. opak:rezerwa, platynka:rezerwa';
AsProgramDescription[8] := '9. opak:220601(200ml), platynka:240234(~ mm)';
AsProgramDescription[9] := '10. opak:220395(shine), platynka:soraya 240965(57mm)';
AsProgramDescription[10] := '11. opak:rezerwa, platynka:rezerwa';
AsProgramDescription[11] := '12. opak:rezerwa, platynka:rezerwa';
AsProgramDescription[12] := '13. opak:rezerwa, platynka:rezerwa';
AsProgramDescription[13] := '14. opak:rezerwa, platynka:rezerwa';
AsProgramDescription[14] := '15. opak:rezerwa, platynka:rezerwa';
END_ACTION

ACTION ResetCommands:

bStepModeMoving 			:= FALSE;
bHeightMotorDown			:= FALSE;
bHeightMotorUp				:= FALSE;
bManualHeightMotorUp		:= FALSE;
bManualHeightMotorDown		:= FALSE;
END_ACTION

ACTION Running:

//Timery
tofMotorUpPermition		(IN:=	bHeightMotorDown,								PT:=T#250MS);
tofMotorDownPermition	(IN:=	bHeightMotorUp,									PT:=T#250MS);
tonTriggerDelay			(IN:=	eRunningState=E_CheckerState.eFormPresent,		PT:=T#50MS);
tonNotBusyDelay			(IN:=	tonTriggerDelay.Q AND NOT bCameraBusy,
																				PT:=T#50MS);
tonLidNOK				(IN:=	eRunningState=E_CheckerState.eFormPresent,
																				PT:=T#50MS);				

CASE eRunningState OF
	
	E_CheckerState.eDisabled:
	
		eRunningState		:=	E_CheckerState.eReady;
	
	//SPRAWDZANIEGOTOWY DO PRACY
	E_CheckerState.eReady:
		
		IF bRun THEN
			eRunningState	:=	E_CheckerState.eFormPresent;	
		END_IF

	//WYKRYTO SLOIK
	E_CheckerState.eFormPresent:
	
		bCameraTrigger		:= TRUE;
		IF	tonTriggerDelay.Q THEN
			IF tonNotBusyDelay.Q AND bCameraGood THEN
				eRunningState	:=	E_CheckerState.eLidOK;		
			ELSIF tonNotBusyDelay.Q  THEN
				eRunningState	:=	E_CheckerState.eLidNOK;	
			END_IF	
		END_IF
		
	
	//BUTELKA W FORMATCE
	E_CheckerState.eBottleOK:
	;
	
	//PLATYNKA OK
	E_CheckerState.eLidOK:
	
		bCheckOK	:= TRUE;
		bCycleDone	:= TRUE;	
	
	//PLATYNKA NOK
	E_CheckerState.eLidNOK:

		bCheckOK	:= FALSE;	
		bCycleDone	:= TRUE;
		
	//NASADKA OK
	E_CheckerState.eCapOK:
	;
		
	//NASADKA NOK
	E_CheckerState.eCapNOK:
	;		

	E_CheckerState.eChecking:
	;
		
END_CASE
END_ACTION

ACTION Statistics:

rtrigCycleTimerRead(CLK:=eRunningState=E_CheckerState.eLidOK OR eRunningState=E_CheckerState.eLidNOK);
IF rtrigCycleTimerRead.Q THEN
		tCycleTime:=tonCycleTimer.ET;
END_IF
tonCycleTimer(IN:=eState>E_Station.eReady,PT:=T#1D);
END_ACTION

END_FUNCTION_BLOCK

// ---- POUs/P07_CapPusher.TcPOU
(*
Nazwa:			P07_CapPusher
Opis:			Wvijak nasadek z sorteram wibracyjnym
Wersja:			v0.1
Data:			2025-11-03
Autor:			DP
Urzadzenia:		
Konfiguracja:	
Info:
- 
*)
PROGRAM P07_CapPusher
VAR_INPUT
	//Szlaban
	//...
	
	//Podajnik
	//...
	
	//Zakrecanie
	//..

END_VAR
VAR
	(*****************SZLABAN*******************)
	fbCapPusherGate										: FB_SpringGateV2;
	QbCapPusherGate										AT %Q*: BOOL; 			// Wyjście sterujące 

	(*******************PODAJNIK*********************)
	fbCapPusherFeeder									: FB_CapPusherFeeder;
	fbCapPusherFeederState								: FB_State;	
	eCapPusherFeederState								: E_Station;
	eCapPusherFeederRunningState						: E_CapFeederState; 	// Stan pracy 
	QbCapPusherFeederSorterVibrator 					AT %Q*: BOOL; 			// Wyjście sterujące 
	QbCapPusherFeederSorterVibrator2 					AT %Q*: BOOL; 			// Wyjście sterujące 	
	QbCapPusherFeederSorterAir 							AT %Q*: BOOL; 			// Wyjście sterujące 
	IbCapPusherFeederHopperSensor						: BOOL; 					
	IbCapPusherFeederWheelSensor						: BOOL; 			
	IbCapPusherFeederSleeveSensor					: BOOL; 
	QnCapPusherFeederVelocitySV 						AT %Q*: UDINT; 			// Nastawa prędkości
	InCapPusherFeederVelocityCV 						AT %I*: UDINT;		
	InCapPusherFeederSTW 								AT %I*: UINT; 			// Statusword transportera wejściowo wyjściowego
	QnCapPusherFeederCTW 								AT %Q*: UINT;  			// Controlword transportera we/wy
	IbCapPusherFeederWcState							AT %I*: BOOL; 			// Statusword transportera wejściowo wyjściowego
	TimerCapPusherFeederEnable							: TOF;
	rtCapPusherFeederEnable								: R_TRIG;
	tonCapPusherFeederEnable							: TON;
	
	(*******ZAKRECANIE**********)
	fbCapPusher											: FB_CapPusher;
	fbCapPusherState									: FB_State;	
	eCapPusherState										: E_Station;
	eCapPusherRunningState								: E_GripperScrewer; 	// Stan pracy 	

	QbCapPusher											AT %Q*: BOOL; 	
	QbCapPusherBlockActuator							AT %Q*: BOOL; 	
	QbCapPusherFormPositioning							AT %Q*: BOOL; 	
	
	IbCapPusherFormSensor								: BOOL; 
	IbCapPusherCapSensor								: BOOL; 
	IbCapPusherUpSensor									: BOOL; 
	IbCapPusherDownSensor								: BOOL; 
	IbCapPusherBlockActuatorOnSensor					: BOOL; 
	IbCapPusherBlockActuatorOffSensor					: BOOL; 
	IbCapPusherFormPositioningUpSensor					: BOOL; 
	IbCapPusherFormPositioningDownSensor				: BOOL; 
	TimerCapPusherEnable								: TOF;
	rtCapPusherEnable									: R_TRIG;
	tonCapPusherEnable									: TON;
	
	(*RFID*)
	//Przed
	bReadedCard 										: BOOL;				
	nReadedCard											: ULINT;	
	fbReader   											: FB_IfmIoLinkRfid;
	AusiReaderInputData  								AT %I* : ARRAY[0..27] OF USINT;
	IbReaderTagPresent									AT %I* : BOOL;
	IBReaderErrorValue									AT %I* : BYTE;
	IbReaderCmdEnd										AT %I* : BOOL;
	IBReaderDataCounterIn								AT %I* : BYTE;
	IbReaderCmdStartAck									AT %I* : BOOL;
	IbReaderCmdStart									AT %Q* : BOOL;
	IBReaderCmmandValue									AT %Q* : BYTE;
	IBReaderDataCounterOut								AT %Q* : BYTE;
	AusiReaderOutputData  								AT %Q* : ARRAY[0..27] OF USINT;	

	(*Lampy*)
	QbCapPusherRedSignalizationLamp 					AT %Q* : BOOL;				
	QbCapPusherGreenSignalizationLamp 					AT %Q* : BOOL;					
	QbCapPusherYellowSignalizationLamp 					AT %Q* : BOOL;							
	
	(*Przyciski*)

	(*Safety*)
		

	QbCapPusherDoors0Close								AT %Q* :BOOL;		// Rozkaz zamkniecia 
	
	(*Zawór główny*)
	QbCapPusherCompressedAir							AT %Q*		:BOOL;		
	IbCapPusherCompressedAirOK 							AT %I*		:BOOL;		//Zasilanie powietrzem sprężonym OK	
	
	(*Zasilanie*)
	IbCapPusherFuseFB1OK								AT %I* :BOOL;		//		
	IbCapPusherFuseFB2OK								AT %I* :BOOL;		//	
	IbCapPusherFuseFB3OK								AT %I* :BOOL;		//	
	
	(*DI wyspy pneumatycznej*)
	QABPneumaticCapPusherEB1ValveCoils 						AT %Q* 	: ARRAY[1..5] OF BYTE;	
	IABPneumaticCapPusherEB1DigitalInput 					AT %I* 	: ARRAY[1..4] OF BYTE;
	IuiPneumaticCapPusherEB1State							AT %I* 	: UINT;	

	(*Czujniki formatek*)
	IbCapPusherThirdFormSensor	 							: BOOL; 		// Czujnik dojazdu 3 formatki
	
	(*Manual*)
	
	(****Inne***)

	
END_VAR

aPowerSupply();
aButtons();
aPneumatics();
aRFID();
aRFID_FB();
aSafety();
aSignalization();
aLimits();
a1_Gate();
a1_GateTime();
a2_Feeder();
a3_Capping();
aWarnings();

(*BAZOWANIE - ZMIAN*)
//SSzlaban
//...
//Podajnik
tonCapPusherFeederEnable (IN:=bCapPusherEnable,PT:=T#5S); 
rtCapPusherFeederEnable(CLK:=tonCapPusherFeederEnable.Q,Q=>);
IF rtCapPusherFeederEnable.Q AND (P00_PackML.fbPMLAuto.ePMLState = E_PMLState.ePMLState_IDLE OR P00_PackML.fbPMLAuto.ePMLState = E_PMLState.ePMLState_EXECUTE)   THEN
	VIS_CP.bCapPusherFeederHeightSet:=TRUE;
ELSIF fbCapPusherFeeder.eState=E_Station.eHomingDone	OR	VIS.bErrorOccure THEN
 	VIS_CP.bCapPusherFeederHeightSet:=FALSE;
END_IF
//Zakrecanie
tonCapPusherEnable (IN:=bCapPusherEnable,PT:=T#5S); 
rtCapPusherEnable(CLK:=tonCapPusherEnable.Q,Q=>);
IF rtCapPusherEnable.Q AND (P00_PackML.fbPMLAuto.ePMLState = E_PMLState.ePMLState_IDLE OR P00_PackML.fbPMLAuto.ePMLState = E_PMLState.ePMLState_EXECUTE)   THEN
	VIS_CP.bCapPusherHeightSet:=TRUE;
ELSIF fbCapPusher.eState=E_Station.eHomingDone	OR	VIS.bErrorOccure THEN
 	VIS_CP.bCapPusherHeightSet:=FALSE;
END_IF
(*KONIEC BAZOWANIE - ZMIANA*)

(*Opoznienie wyłączanie enabla*)
//Szlaban
//..
//Podajnik
TimerCapPusherFeederEnable	(IN:=bCapPusherEnable,	PT:=T#2S);
//Zakrecanie
TimerCapPusherEnable		(IN:=bCapPusherEnable, PT:=T#2S);

(*Staty*)
//Szlaban
//...
//Podajnik
fbCapPusherFeederState(
	eState							:=	eCapPusherFeederState , 
	bRun							:=	VIS_CP.bCapPusherFeederRun,	
	eCapFeederRunningState			:=	eCapPusherFeederRunningState , 
	sStateDesc						=>	VIS_CP.sCapPusherFeederState,
	iState							=>	VIS_CP.iCapPusherFeederState);	

//Zakrecanie
fbCapPusherState(
	eState							:=	eCapPusherState , 
	bRun							:=	VIS_CP.bCapPusherRun,	
	eGripperScrewerRunningState		:=	eCapPusherRunningState , 
	sStateDesc						=>	VIS_CP.sCapPusherState,
	iState							=>	VIS_CP.iCapPusherState);	


(********KASOWANIE ROZKAZÓW CYKLI*********)
//Szlaban
//...
//Podajnik
//...
//Zakrecanie
IF fbCapPusher.bCycleDone1 AND bManualMode THEN
	VIS_CP.bCapPusherRun 		:= FALSE;
END_IF

ACTION a1_Gate:
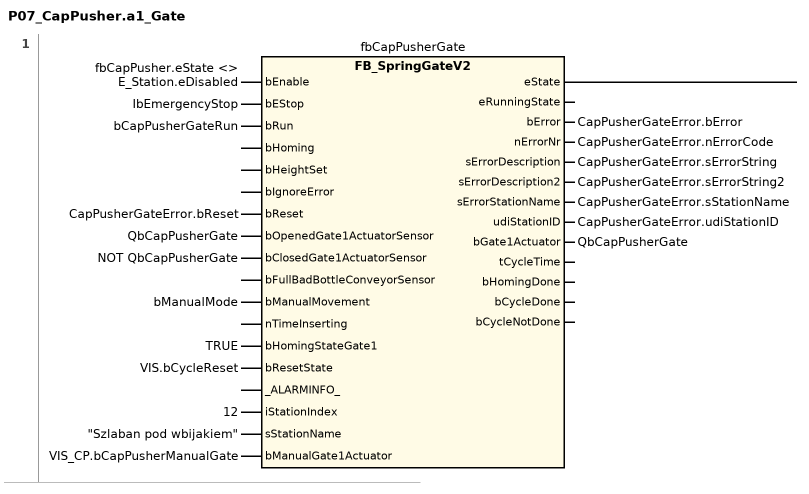
// NETWORK 1
fbCapPusherGate(
    bEnable := fbCapPusher.eState <> E_Station.eDisabled,
    bEStop := IbEmergencyStop,
    bRun := bCapPusherGateRun,
    bReset := CapPusherGateError.bReset,
    bOpenedGate1ActuatorSensor := QbCapPusherGate,
    bClosedGate1ActuatorSensor := NOT QbCapPusherGate,
    bManualMovement := bManualMode,
    bHomingStateGate1 := TRUE,
    bResetState := VIS.bCycleReset,
    iStationIndex := 12,
    sStationName := "Szlaban pod wbijakiem",
    bManualGate1Actuator := VIS_CP.bCapPusherManualGate,
    bError => CapPusherGateError.bError,
    nErrorNr => CapPusherGateError.nErrorCode,
    sErrorDescription => CapPusherGateError.sErrorString,
    sErrorDescription2 => CapPusherGateError.sErrorString2,
    sErrorStationName => CapPusherGateError.sStationName,
    udiStationID => CapPusherGateError.udiStationID,
    bGate1Actuator => QbCapPusherGate); // FB_SpringGateV2
END_ACTION

ACTION a1_GateTime:

fbCapPusherGate.nTimeInserting	:=	300;
END_ACTION

ACTION a2_Feeder:
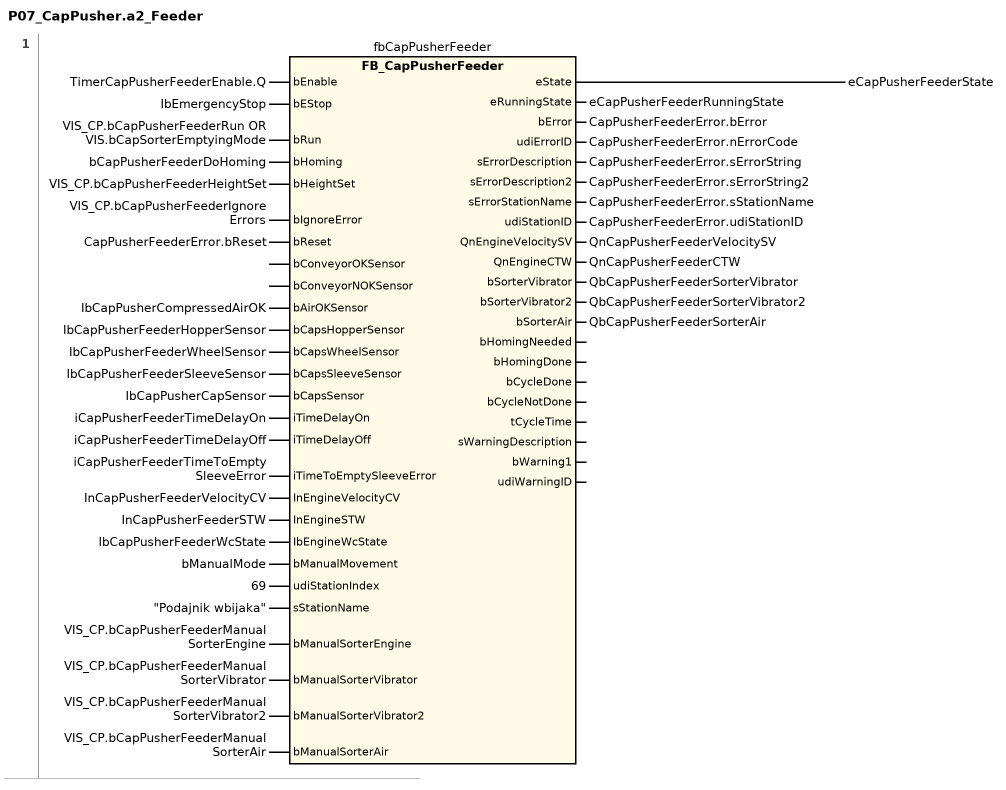
// NETWORK 1
fbCapPusherFeeder(
    bEnable := TimerCapPusherFeederEnable.Q,
    bEStop := IbEmergencyStop,
    bRun := VIS_CP.bCapPusherFeederRun OR VIS.bCapSorterEmptyingMode,
    bHoming := bCapPusherFeederDoHoming,
    bHeightSet := VIS_CP.bCapPusherFeederHeightSet,
    bIgnoreError := VIS_CP.bCapPusherFeederIgnoreErrors,
    bReset := CapPusherFeederError.bReset,
    bAirOKSensor := IbCapPusherCompressedAirOK,
    bCapsHopperSensor := IbCapPusherFeederHopperSensor,
    bCapsWheelSensor := IbCapPusherFeederWheelSensor,
    bCapsSleeveSensor := IbCapPusherFeederSleeveSensor,
    bCapsSensor := IbCapPusherCapSensor,
    iTimeDelayOn := iCapPusherFeederTimeDelayOn,
    iTimeDelayOff := iCapPusherFeederTimeDelayOff,
    iTimeToEmptySleeveError := iCapPusherFeederTimeToEmptySleeveError,
    InEngineVelocityCV := InCapPusherFeederVelocityCV,
    InEngineSTW := InCapPusherFeederSTW,
    IbEngineWcState := IbCapPusherFeederWcState,
    bManualMovement := bManualMode,
    udiStationIndex := 69,
    sStationName := "Podajnik wbijaka",
    bManualSorterEngine := VIS_CP.bCapPusherFeederManualSorterEngine,
    bManualSorterVibrator := VIS_CP.bCapPusherFeederManualSorterVibrator,
    bManualSorterVibrator2 := VIS_CP.bCapPusherFeederManualSorterVibrator2,
    bManualSorterAir := VIS_CP.bCapPusherFeederManualSorterAir,
    eRunningState => eCapPusherFeederRunningState,
    bError => CapPusherFeederError.bError,
    udiErrorID => CapPusherFeederError.nErrorCode,
    sErrorDescription => CapPusherFeederError.sErrorString,
    sErrorDescription2 => CapPusherFeederError.sErrorString2,
    sErrorStationName => CapPusherFeederError.sStationName,
    udiStationID => CapPusherFeederError.udiStationID,
    QnEngineVelocitySV => QnCapPusherFeederVelocitySV,
    QnEngineCTW => QnCapPusherFeederCTW,
    bSorterVibrator => QbCapPusherFeederSorterVibrator,
    bSorterVibrator2 => QbCapPusherFeederSorterVibrator2,
    bSorterAir => QbCapPusherFeederSorterAir); // FB_CapPusherFeeder
eCapPusherFeederState := fbCapPusherFeeder.eState;
END_ACTION

ACTION a3_Capping:
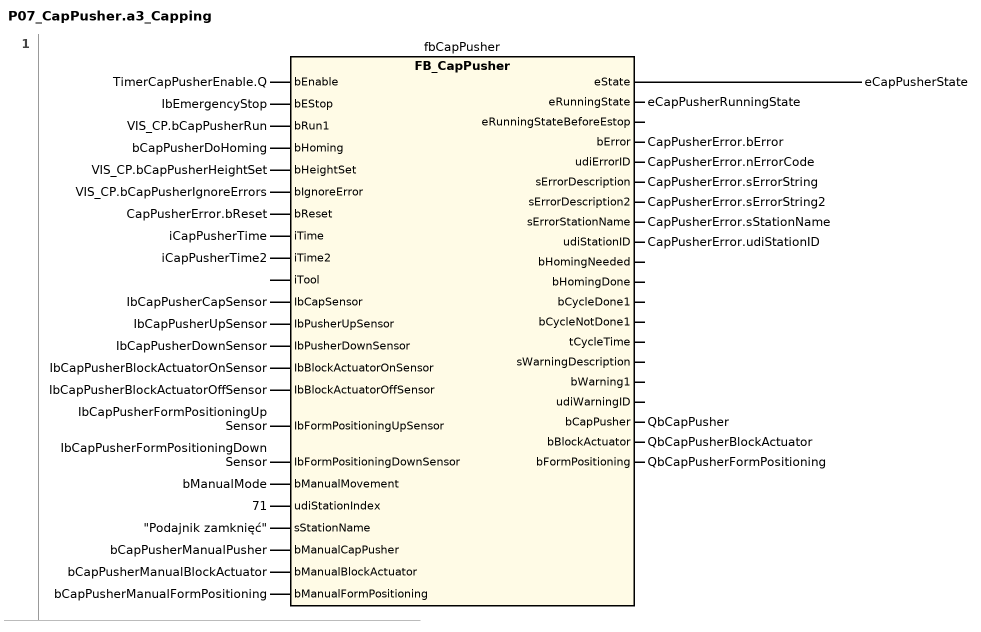
// NETWORK 1
fbCapPusher(
    bEnable := TimerCapPusherEnable.Q,
    bEStop := IbEmergencyStop,
    bRun1 := VIS_CP.bCapPusherRun,
    bHoming := bCapPusherDoHoming,
    bHeightSet := VIS_CP.bCapPusherHeightSet,
    bIgnoreError := VIS_CP.bCapPusherIgnoreErrors,
    bReset := CapPusherError.bReset,
    iTime := iCapPusherTime,
    iTime2 := iCapPusherTime2,
    IbCapSensor := IbCapPusherCapSensor,
    IbPusherUpSensor := IbCapPusherUpSensor,
    IbPusherDownSensor := IbCapPusherDownSensor,
    IbBlockActuatorOnSensor := IbCapPusherBlockActuatorOnSensor,
    IbBlockActuatorOffSensor := IbCapPusherBlockActuatorOffSensor,
    IbFormPositioningUpSensor := IbCapPusherFormPositioningUpSensor,
    IbFormPositioningDownSensor := IbCapPusherFormPositioningDownSensor,
    bManualMovement := bManualMode,
    udiStationIndex := 71,
    sStationName := "Podajnik zamknięć",
    bManualCapPusher := bCapPusherManualPusher,
    bManualBlockActuator := bCapPusherManualBlockActuator,
    bManualFormPositioning := bCapPusherManualFormPositioning,
    eRunningState => eCapPusherRunningState,
    bError => CapPusherError.bError,
    udiErrorID => CapPusherError.nErrorCode,
    sErrorDescription => CapPusherError.sErrorString,
    sErrorDescription2 => CapPusherError.sErrorString2,
    sErrorStationName => CapPusherError.sStationName,
    udiStationID => CapPusherError.udiStationID,
    bCapPusher => QbCapPusher,
    bBlockActuator => QbCapPusherBlockActuator,
    bFormPositioning => QbCapPusherFormPositioning); // FB_CapPusher
eCapPusherState := fbCapPusher.eState;
END_ACTION

ACTION aButtons:

END_ACTION

ACTION aLimits:
(*
Nazwa:			aLimits
Opis:			Zabezpieczenia
Wersja:			v1.0
Data:			2023-11-24
Autor:			DP
Urzadzenia:		
Zmiany:	

Info:
*)

(**** Limity i zabezpieczenia***)
END_ACTION

ACTION aPneumatics:
// Do podpięcia według kolejności
QbCapPusherGate;
QbCapPusherFeederSorterAir;
QbCapPusher;			
QbCapPusherBlockActuator;	
QbCapPusherFormPositioning;

(*************************** CapPusher EB1 **************************************)
// Wyspa 1 - dozowanie
IuiPneumaticCapPusherEB1State;
QABPneumaticCapPusherEB1ValveCoils[1].0	:= QbCapPusher;
QABPneumaticCapPusherEB1ValveCoils[1].1 := NOT QbCapPusher;
QABPneumaticCapPusherEB1ValveCoils[1].2 := QbCapPusherBlockActuator;
QABPneumaticCapPusherEB1ValveCoils[1].3 ;
QABPneumaticCapPusherEB1ValveCoils[1].4 := QbCapPusherFormPositioning;
QABPneumaticCapPusherEB1ValveCoils[1].5 ;
QABPneumaticCapPusherEB1ValveCoils[1].6 := NOT QbCapPusherGate;
QABPneumaticCapPusherEB1ValveCoils[1].7 := QbCapPusherGate; 
QABPneumaticCapPusherEB1ValveCoils[2].0 ;				
QABPneumaticCapPusherEB1ValveCoils[2].1 ;
QABPneumaticCapPusherEB1ValveCoils[2].2 ;
QABPneumaticCapPusherEB1ValveCoils[2].3 ;
QABPneumaticCapPusherEB1ValveCoils[2].4 ;											
QABPneumaticCapPusherEB1ValveCoils[2].5 ;
QABPneumaticCapPusherEB1ValveCoils[2].6 ;
QABPneumaticCapPusherEB1ValveCoils[2].7 ;
QABPneumaticCapPusherEB1ValveCoils[3].0 ;
QABPneumaticCapPusherEB1ValveCoils[3].1 ;
QABPneumaticCapPusherEB1ValveCoils[3].2 ;
QABPneumaticCapPusherEB1ValveCoils[3].3 ;
QABPneumaticCapPusherEB1ValveCoils[3].4 ; 
QABPneumaticCapPusherEB1ValveCoils[3].5 ;
QABPneumaticCapPusherEB1ValveCoils[3].6 ;
QABPneumaticCapPusherEB1ValveCoils[3].7 ;                                               
QABPneumaticCapPusherEB1ValveCoils[4].0	;		                                
QABPneumaticCapPusherEB1ValveCoils[4].1 ;                                       
QABPneumaticCapPusherEB1ValveCoils[4].2	;		                                
QABPneumaticCapPusherEB1ValveCoils[4].3 ;                                      
QABPneumaticCapPusherEB1ValveCoils[4].4 ;		                                
QABPneumaticCapPusherEB1ValveCoils[4].5 ;        
QABPneumaticCapPusherEB1ValveCoils[4].6 ;		
QABPneumaticCapPusherEB1ValveCoils[4].7 ; 
                                                              
(*********************Koniec CapPusher EB1 **************************************) 


//Zawór głównego powietrza
QbCapPusherCompressedAir	:=	IbEmergencyStop AND QbCapPusherFeederSorterAir;

(*************************** EB1 **************************************)
// Wyspa 1 - 52N8
IuiPneumaticCapPusherEB1State;
//DI1
IbCapPusherFeederHopperSensor		:=	IABPneumaticCapPusherEB1DigitalInput[1].0;	
IbCapPusherFeederWheelSensor		:=	NOT IABPneumaticCapPusherEB1DigitalInput[1].1;	
IbCapPusherFeederSleeveSensor		:=	IABPneumaticCapPusherEB1DigitalInput[1].2;	
										IABPneumaticCapPusherEB1DigitalInput[1].3;
IbCapPusherUpSensor					:=	IABPneumaticCapPusherEB1DigitalInput[1].4;	
IbCapPusherDownSensor				:=	IABPneumaticCapPusherEB1DigitalInput[1].5;	
IbCapPusherCapSensor				:=	IABPneumaticCapPusherEB1DigitalInput[1].6;	
										;IABPneumaticCapPusherEB1DigitalInput[1].7;	
//DI2                                           
IbCapPusherBlockActuatorOffSensor	:=	IABPneumaticCapPusherEB1DigitalInput[2].0;	
IbCapPusherBlockActuatorOnSensor	:=	IABPneumaticCapPusherEB1DigitalInput[2].1;	
IbCapPusherFormSensor				:=	IABPneumaticCapPusherEB1DigitalInput[2].2;	
IbCapPusherFormPositioningDownSensor:=	IABPneumaticCapPusherEB1DigitalInput[2].3;	
IbCapPusherFormPositioningUpSensor	:=	IABPneumaticCapPusherEB1DigitalInput[2].4;	
;	IABPneumaticCapPusherEB1DigitalInput[2].5;		
;	IABPneumaticCapPusherEB1DigitalInput[2].6;		
;	IABPneumaticCapPusherEB1DigitalInput[2].7;	

// Wyspa 1 - 52N8A
IuiPneumaticCapPusherEB1State;
//DI1
;	IABPneumaticCapPusherEB1DigitalInput[3].0;	
;	IABPneumaticCapPusherEB1DigitalInput[3].1;	
;	IABPneumaticCapPusherEB1DigitalInput[3].2;	
;	IABPneumaticCapPusherEB1DigitalInput[3].3;
;	IABPneumaticCapPusherEB1DigitalInput[3].4;	
;	IABPneumaticCapPusherEB1DigitalInput[3].5;		
;	IABPneumaticCapPusherEB1DigitalInput[3].6;		
;	IABPneumaticCapPusherEB1DigitalInput[3].7;
//DI2                                               		
;	IABPneumaticCapPusherEB1DigitalInput[4].0;
;	IABPneumaticCapPusherEB1DigitalInput[4].0;	
;	IABPneumaticCapPusherEB1DigitalInput[4].1;	
;	IABPneumaticCapPusherEB1DigitalInput[4].2;	
;	IABPneumaticCapPusherEB1DigitalInput[4].3;	
;	IABPneumaticCapPusherEB1DigitalInput[4].4;
;	IABPneumaticCapPusherEB1DigitalInput[4].5;		
;	IABPneumaticCapPusherEB1DigitalInput[4].6;		
	IABPneumaticCapPusherEB1DigitalInput[4].7;	
(*********************Koniec EB2 **************************************)
END_ACTION

ACTION aPowerSupply:


	//Dodane do głwnych
	IbCapPusherFuseFB1OK	; //Przekaznik kontroli faz
	IbCapPusherFuseFB2OK	; //Kontrola poprawności faz
	IbCapPusherFuseFB3OK	; //Blok bezpiecznikowy
END_ACTION

ACTION aRFID:
(*Przepisanie bity wykrycia karty*)
bReadedCard 		:= IbReaderTagPresent AND fbReader.bCodeReaded;
nReadedCard 		:= DINT_TO_ULINT(fbReader.diReadedCode);
END_ACTION

ACTION aRFID_FB:
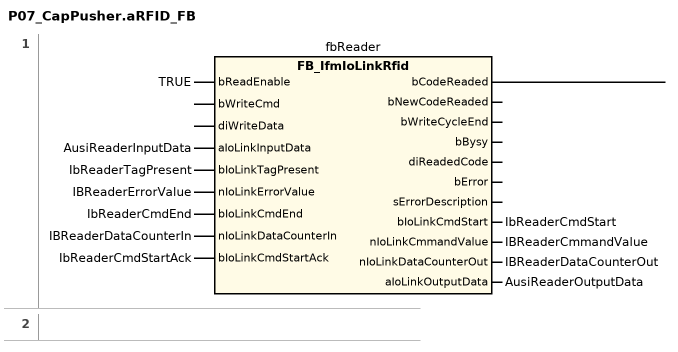
// NETWORK 1
fbReader(
    bReadEnable := TRUE,
    aIoLinkInputData := AusiReaderInputData,
    bIoLinkTagPresent := IbReaderTagPresent,
    nIoLinkErrorValue := IBReaderErrorValue,
    bIoLinkCmdEnd := IbReaderCmdEnd,
    nIoLinkDataCounterIn := IBReaderDataCounterIn,
    bIoLinkCmdStartAck := IbReaderCmdStartAck,
    bIoLinkCmdStart => IbReaderCmdStart,
    nIoLinkCmmandValue => IBReaderCmmandValue,
    nIoLinkDataCounterOut => IBReaderDataCounterOut,
    aIoLinkOutputData => AusiReaderOutputData); // FB_IfmIoLinkRfid

// NETWORK 2
END_ACTION

ACTION aSafety:

// Dodać do P00_Alarms.aGeneralAlarms
	//IbCapPusherEmergencyStopButton0Pressed;
	//IbCapPusherEmergencyStopButton1Pressed;
	
(*
	IF IbCapPusherEmergencyStopButton0Pressed THEN
		GeneralAlarms.nErrorCode:=1;			
		GeneralAlarms.sErrorString:='Stop Awaryjny, sprawdź bezpieczeństwo, zresetuj przyciskiem na panelu | Naciśnięty przycisk awaryjny 1 na CapPusher';	
	ELSIF  IbCapPusherEmergencyStopButton1Pressed THEN
		GeneralAlarms.nErrorCode:=2;
		GeneralAlarms.sErrorString:='Stop Awaryjny, sprawdź bezpieczeństwo, zresetuj przyciskiem na panelu | Naciśnięty przycisk awaryjny 2 na CapPusher';	
*)	
	

// Dodać do miejsca gdzie są zamykane drzwi	
// lub zostawić tak jak jest
	QbCapPusherDoors0Close := QbDispencersDoorsClose;
END_ACTION

ACTION aSignalization:
(*****Listwy LED*****)

QbCapPusherRedSignalizationLamp		:= INT_TO_BOOL(P00_Signalization.QiLineRedSignalizationLamp);
QbCapPusherGreenSignalizationLamp	:= INT_TO_BOOL(P00_Signalization.QiLineGreenSignalizationLamp);
QbCapPusherYellowSignalizationLamp	:= INT_TO_BOOL(P00_Signalization.QiLineBlueSignalizationLamp);


//QbCapPusherStartLamp	:= P00_Signalization.QbStartLamp;	   
//QbCapPusherResetLamp	:= P00_Signalization.QbResetLamp;
END_ACTION

ACTION aWarnings:
//Warning 0
IF fbCapPusherFeeder.bWarning1 AND NOT CapSorterWarning[0].bWarning THEN
	CapSorterWarning[0].bWarning										:=TRUE;
	CapSorterWarning[0].udiWarningCode									:=41;
	CapSorterWarning[0].sDescription									:='Sorter nasadek | Brak nasadek w zasobniku';
ELSIF NOT fbCapPusherFeeder.bWarning1 THEN 
	CapSorterWarning[0].bWarning										:=FALSE;
	CapSorterWarning[0].bAcknowledge									:=FALSE;
	VIS.uliWarningAcknowledge.27										:=FALSE;
ELSIF CapSorterWarning[0].bAcknowledge THEN                               
	CapSorterWarning[0].bAcknowledge									:=TRUE;
END_IF
END_ACTION

END_PROGRAM

// ---- POUs/FB/FB_CapPusherFeeder.TcPOU
(*
Nazwa:			FB_CapPusherFeeder
Opis:			Sorter wibracyjny z rękawem
Wersja:			v1.0
Data:			2025-11-17
Autor:			DP
Urzadzenia:		Wkbracje, Wydmuch, czujniki zapełnienia rękawa
Konfiguracja:	
Info:
-
*)


FUNCTION_BLOCK FB_CapPusherFeeder
VAR_INPUT	
	bEnable						: BOOL;					//Zezowlenie na pracę stacji sprawdzania
	bEStop						: BOOL;					//Stop Awaryjny nieaktywny
	bRun						: BOOL;					//
	bHoming						: BOOL;					//Zezwolenie na wykonanie bazowania i pozycjonowania stacji sprawdzania
	bHeightSet					: BOOL;					//Bit do bazowania stacji na ustaloną wysokość 
	bIgnoreError				: BOOL;					//Ignorowania błędów cyklu pracy
	bReset						: BOOL;					//Reset błędu, jeśli w stanie "eError"

	bConveyorOKSensor			: BOOL;					
	bConveyorNOKSensor			: BOOL;				
	bAirOKSensor				: BOOL;					// 

	bCapsHopperSensor			: BOOL;					// Czujnik poziomu
	bCapsWheelSensor			: BOOL;					// Czujnik poziomu
	bCapsSleeveSensor			: BOOL;					// 
	bCapsSensor					: BOOL;

	iTimeDelayOn				: INT; 					//Czas na właczenie silnika sortera po zaniku sygnału przepełnienia z rękawa
	iTimeDelayOff				: INT; 					// Czas na wylączenie silnika sortera po wykryciu sygnału przepełnienia z rękawa sortera
	iTimeToEmptySleeveError		: INT;					// Czas do włączenia alrmu pustego rękawa
	InEngineVelocityCV 			: UDINT;		
	InEngineSTW 				: UINT; 				// Statusword transportera wejściowo wyjściowego
	IbEngineWcState				: BOOL; 				// Statusword transportera wejściowo wyjściowego

	bManualMovement				: BOOL; 				//Uruchomienie trybu ruchów ręcznych
	udiStationIndex				: UDINT;				// Indywidualny numer stacji
	sStationName				: WSTRING;				// Nazwa stacji	
END_VAR

VAR_OUTPUT
	eState						: E_Station;			// Aktualny stan stacju
	eRunningState				: E_CapFeederState;		// Stan pracy stacji
	bError						: BOOL;					// Błąd stacji
	udiErrorID					: UDINT;				// Nr blędu przeciągania formatek
	sErrorDescription			: STRING(200);			// Opis błędu
	sErrorDescription2			: STRING(200);			// Opis błędu
	sErrorStationName			: STRING;				// Nazwa stacj
	udiStationID				: UDINT;				// Nr stacji

	QnEngineVelocitySV 			: UDINT; 				// Nastawa prędkości
	QnEngineCTW 				: UINT;  				// Controlword transportera we/wy	
	bSorterVibrator				: BOOL; 	
	bSorterVibrator2			: BOOL; 	
	bSorterAir 					: BOOL; 							
	
	bHomingNeeded				: BOOL;					// Wymagane ponowne bazowanie (blad podczas bazowania lub stop awaryjny)
	bHomingDone					: BOOL;					// Stacja zbazowana 
	bCycleDone					: BOOL;					// Sygnał o zakończeniu cyklu
	bCycleNotDone				: BOOL;					// Sygnał o niezakończonym cyklu
	tCycleTime					: TIME;	 				// Czas cyklu 
	sWarningDescription			: STRING;
	bWarning1					: BOOL;
	udiWarningID				: UDINT;
END_VAR

VAR_IN_OUT
	bManualSorterEngine			: BOOL;					//
	bManualSorterVibrator		: BOOL;					//
	bManualSorterVibrator2		: BOOL;					//
	bManualSorterAir 			: BOOL;					//
END_VAR

VAR
	i							:	INT;

	// State
	eLastState					: E_Station;			//Stan ogólny bloku
	eLastStateTemp				: E_Station;			//Stan ogólny bloku
	eLastRunningState			: E_CapFeederState;		//Stan podbloku
	eLastRunningStateTemp		: E_CapFeederState;		//Stan podbloku

	bStateError					: BOOL;
		
	tonSortingEngineOn			: TON;					// Opóźnienie po załączeniu napędu
	tonSortingEngineOff			: TON;					// Opóźnienie wyłączenia napędu
	tonAirBeforeStart			: TON;					// Czasówka opóźeniani przedmuchu
	tonAirAfterStop				: TON;					// Czasówka przedmuchu po zatrzymaniu
	tonStoppingTime				: TON;					// Czasówka zbyt długiego zatrzymawania

	tonEmptySleeveError			: TON;					// Timer pustego rękawa
	tonCycleTimer				: TON;					// Czasówka cyklu
	rtrigCycleTimerRead			: R_TRIG;				// Trigger do statystyk cyklu 
	
	fbInverter: FB_MitsubishiInverter;
	tonInverterError: TON;
	tonAirError: TON;
	(*Ostrzeżenia*)
	fbbLevelSensor:	FB_InputFilter_v2;
	(*Inne*)	
	fbbCapsWheelLevelSensor 		: FB_InputFilter_v2;
	fbbCapsAndSleeveSensor			: FB_InputFilter_v2;
	tonVibrator2AndNotbCapsSensor	: TON;
	tonbSorterVibrator				: TON;
	tonfbInverterbRun1				: TON;
	tonfbInverterbRun2				: TON;	
	//Zmienne od EVENTLOGGER
	bAlarmInit 						: BOOL := TRUE; 
	nAlarmNumerator					: INT;
	arfbAlarm						: ARRAY[0..19] OF  FB_TcAlarm;		//Tablica bloczków błędów
	fbSourceInfo 					: FB_TcSourceInfo;
	iSourceInfo						: I_TcSourceInfo;
	sAlarmTest						: STRING;
	//Koniec zmiennych od EVENTLOGGER
	iSortingCASE					: INT;
	tonNoCapsHopperSensor			: TON;
END_VAR

//Wywołanie bloczków od stacji. Ważna jest ich kolejność!!!
ACT_Limits();
ACT_ErrorHandling();
ACT_Signals();
ACT_Control();
ACT_Inverter();
ACT_Statistic();
ACT_Status();
ACT_Warnings();
aStationID();

ACTION ACT_Control:
	(*****Wyłączenie enable*****)
	IF NOT bEnable THEN
		IF eState <> E_Station.eDisabled AND eState <> E_Station.ePreparingToDisable THEN
				eState 				:= E_Station.ePreparingToDisable; 
		END_IF	
	END_IF

	(*****Estop*****)
	IF NOT bEstop  THEN	
		IF eState <> E_Station.eAborted AND eState <> E_Station.eAborting AND eState <> E_Station.eDisabled THEN
				eState 				:= E_Station.eAborting; 
		END_IF
	END_IF

	CASE eState OF
//--------------------------------------------------------------------------------
// Stan maszyny po wyłączeniu i przygotowanie do uruchomienia
	E_Station.eDisabled: 					// Stan nieaktywnosci (Stacja wyłączona) 
	
		IF bEnable THEN
			eState 				:= E_Station.ePreparingToReady; 
		END_IF 
		
//--------------------------------------------------------------------------------
// Stan maszyny po zatrzymaniu awaryjnym   
	E_Station.eAborted: 					// Stan bezpiecznego zatrzymania (po Abortingu) 

		IF bEStop THEN
			eState 				:= E_Station.ePreparingToReady;
		END_IF
		
//--------------------------------------------------------------------------------
// Stan maszyny naciśnieciu estopa 	
	E_Station.eAborting:                 	// Stan bezpiecznego zatrzymywania (po EStopie)

		ACT_ResetCommands();

		eState 						:=  E_Station.eAborted;  
		eRunningState				:=	E_CapFeederState.eReady;
		
//--------------------------------------------------------------------------------
// Stan masyzny po wykryciu błędu			
	E_Station.eError:                 	 	// Stan błędu 	
		
		ACT_ResetCommands();
		
		IF bReset THEN
			eState 				:= E_Station.eResetting;
			bError				:= FALSE;
		END_IF
		
//--------------------------------------------------------------------------------
// Stan masyzny po wykryciu błędu
	E_Station.eResetting:					// Stan resetowania bledu (po Errorze)
		
			fbInverter.bReset	:= TRUE;
		IF NOT bError (*AND fbInverter.eState = E_Station.eReady*) THEN
			fbInverter.bReset	:= FALSE;	
			//{warning 'Sprawdzić błąd falownika CapFeeder'}
			udiErrorID 			:=	0;
			sErrorDescription 	:=	'';
			eState 				:=	E_Station.ePreparingToReady;
			eRunningState		:=	E_CapFeederState.eReady;
		ELSE
			eState 				:=	E_Station.eError;
		END_IF
    
//--------------------------------------------------------------------------------
// Stan ruchoow manualnych
	E_Station.eManualMovement:     			// Stan ruchów manualnych  
   
		ACT_ManualMovements();
		//Wyjście z trybu serwisowego
		IF NOT bManualMovement THEN		
			eState:=E_Station.eReady;
		END_IF
		

//--------------------------------------------------------------------------------
// Stan rozpoczecia bazowania
	E_Station.eHoming:						// Stan bazowania 
		
		ACT_Homing();
		IF NOT bHoming AND NOT bHeightSet THEN
		   eState								:=	E_Station.ePreparingToReady;
		END_IF		
		
//--------------------------------------------------------------------------------
// Stan zakończenia bazowania
	E_Station.eHomingDone:                  // Stan wykonania bazowania 
	
		bHomingDone							:=	TRUE;
		IF NOT bHoming AND NOT bHeightSet THEN
		   eState:=E_Station.eReady;
		END_IF
		
//--------------------------------------------------------------------------------
// Stan przygotowania do gotowości
	E_Station.ePreparingToReady:            // Stan przygotowywania do gotowosci (zawsze przed Ready)  
		
		fbInverter.bRun						:=	FALSE;
		bSorterAir							:=	FALSE;
		bSorterVibrator						:=	FALSE;
		bSorterVibrator2					:=	FALSE;

		eRunningState						:=	E_CapFeederState.eReady;
		eState								:=	E_Station.eReady;	
		
//-------------------------------------------------------------------------------
// Stan przygotowania do wyłączenia maszyny
	E_Station.ePreparingToDisable:          // Stan przygotowywania do nieaktywnosci (po wyłączeniu Enable) 
		
		bSorterAir							:=	FALSE;

		eRunningState						:=	E_CapFeederState.eReady;		
		eState								:=	E_Station.eDisabled;

			
//--------------------------------------------------------------------------------
// Stan gotowości
	E_Station.eReady:						// Stan gotowosci 

		IF bRun AND NOT bCycleDone AND NOT bCycleNotDone THEN
			eState 							:= E_Station.eStarting; 
		END_IF
		IF bHoming OR bHeightSet THEN
			bHomingDone						:=	FALSE;
			eState 							:=	E_Station.eHoming; 
		END_IF
		IF bManualMovement THEN
			//Jeśli przejście w tryb ruchów manualnych przepisz wszystkie stany siłowników sterowanych przez moduł
			//aby zapobiec ewentualnym kolizjom po wejściu w tryb serwisowy
			eState 						:= E_Station.eManualMovement; 
		END_IF
		IF NOT bRun THEN
			bCycleDone 			:= FALSE;
			bCycleNotDone 		:= FALSE;			
		END_IF
		
//--------------------------------------------------------------------------------
// Stan zatrzymywania
	E_Station.eStopping:					// Stan zatrzymywania 
		
	bSorterVibrator	:=	FALSE;
	bSorterVibrator2:=	FALSE;
	bSorterAir		:=	TRUE;
	fbInverter.bRun := FALSE;
	
	IF tonStoppingTime.Q THEN
		ACT_ResetCommands();
		eRunningState							:= E_CapFeederState.eReady;
		eState									:= E_Station.eReady;
	END_IF
		
//--------------------------------------------------------------------------------
// Stan uruchomienia lini ( po eReady)
	E_Station.eStarting:                  	// Stan uruchamiania (po Ready)

		eState					 := E_Station.eRunning; 
		
//--------------------------------------------------------------------------------
// Stan wykonywania pracy
	E_Station.eRunning:               		// Stan wykonywania cyklu (po Startingu), w tym stanie osobny

		ACT_Running();
		IF NOT bRun THEN 					(*Przerywanie cyklu*)
			eState				:= E_Station.eStopping;
			//bCycleNotDone		:= TRUE;
		END_IF
		(*IF bCycleDone OR bCycleNotDone THEN (*Cykl zakończony*)
			eState 				 := E_Station.eReady;
		END_IF*)							
		
END_CASE
END_ACTION

ACTION ACT_ErrorHandling:
// Alarm_0600	600	Error	Pusty rekaw wbijaka nasadek - sprawdź czy nasadki sie nie zablokowały
// Alarm_0601	601	Error	Błąd falownika - możliwe zablokowanie mechaniczne transportera
// Alarm_0602	602	Error	Bład czujnika powietrza - sprwadź ciśnienie

IF bAlarmInit THEN
    bAlarmInit := FALSE; 
	fbSourceInfo.Clear();
	fbSourceInfo.sName:=wsLiteral_TO_UTF8(sStationName);//'Machine';
	fbSourceInfo.nId:=udiStationID;//2700;
	// Alarm_0600	600	Error	Pusty rekaw wbijaka nasadek - sprawdź czy nasadki sie nie zablokowały
    arfbAlarm[0].CreateEx(stEventEntry := TC_EVENTS.AlarmClass.Alarm_0600, bWithConfirmation:= FALSE,  ipSourceInfo:= fbSourceInfo); 
	// Alarm_0601	601	Error	Błąd falownika - możliwe zablokowanie mechaniczne transportera
	arfbAlarm[1].CreateEx(stEventEntry := TC_EVENTS.AlarmClass.Alarm_0601, bWithConfirmation:= FALSE,  ipSourceInfo:= fbSourceInfo);
	// Alarm_0602	602	Error	Bład czujnika powietrza - sprwadź ciśnienie	
	arfbAlarm[2].CreateEx(stEventEntry := TC_EVENTS.AlarmClass.Alarm_0602, bWithConfirmation:= FALSE,  ipSourceInfo:= fbSourceInfo);	
	// Alarm_0603	603	Error	Blokada nasadek przed wbijaniem - sprawdź czujnik
    arfbAlarm[3].CreateEx(stEventEntry := TC_EVENTS.AlarmClass.Alarm_0603, bWithConfirmation:= FALSE,  ipSourceInfo:= fbSourceInfo);  
	// Alarm_0604	604	Error	Brak nakrętek w zbiorniku
    arfbAlarm[4].CreateEx(stEventEntry := TC_EVENTS.AlarmClass.Alarm_0604, bWithConfirmation:= FALSE,  ipSourceInfo:= fbSourceInfo);	{warning 'Zmienić opis alarmu powyżej po dodaniu do listy'}
END_IF

//OBSŁUGA BŁĘDÓW STACJI SPRAWDZANIA
//************LISTA BŁĘDÓW***************
bStateError:= (eState=E_Station.eError) OR (eState=E_Station.eResetting);

//************LISTA BŁĘDÓW***************

//Error 1 - podnośnik nie porusza się pomimo wysterowania 
tonEmptySleeveError				(IN:=NOT bCapsSleeveSensor AND bRun, PT:=INT_TO_TIME(iTimeToEmptySleeveError)*1000); //Było 30, teraz jest z receptur
tonInverterError				(IN:=fbInverter.bError AND NOT bStateError, PT:=T#3S);
tonAirError						(IN:=bSorterAir AND NOT bAirOKSensor AND NOT bStateError, PT:=T#3S);
tonVibrator2AndNotbCapsSensor	(IN:=bSorterVibrator2 AND fbbCapsWheelLevelSensor.bOut AND  NOT bCapsSensor AND P07_CapPusher.fbCapPusherFeeder.eState = E_Station.eRunning, PT:=T#30S);
tonNoCapsHopperSensor			(IN:= NOT bCapsHopperSensor AND P07_CapPusher.fbCapPusherFeeder.eState = E_Station.eRunning AND NOT VIS.bConfectionEnding, PT:=T#30S);

IF (bEnable OR (eState = E_Station.ePreparingToDisable)) THEN
	
		
	//Error - Pusty rekaw sortera nasadek
	IF tonEmptySleeveError.Q THEN
		IF NOT arfbAlarm[0].bActive THEN
			arfbAlarm[0].Raise(nTimeStamp:=0);
		END_IF
	ELSE	
		IF  arfbAlarm[0].bActive AND bReset THEN
			arfbAlarm[0].Clear(nTimeStamp:=0, bResetConfirmation:= FALSE);
		END_IF
	END_IF	
		
	//Error - Bład falownika
	IF tonInverterError.Q THEN
		IF NOT arfbAlarm[1].bActive THEN
			arfbAlarm[1].Raise(nTimeStamp:=0);
		END_IF
	ELSE	
		IF  arfbAlarm[1].bActive AND bReset THEN
			arfbAlarm[1].Clear(nTimeStamp:=0, bResetConfirmation:= FALSE);
		END_IF
	END_IF		
	
	//Error - Bład powietrza
	IF tonAirError.Q THEN
		IF NOT arfbAlarm[2].bActive THEN
			arfbAlarm[2].Raise(nTimeStamp:=0);
		END_IF
	ELSE	
		IF  arfbAlarm[2].bActive AND bReset THEN
			arfbAlarm[2].Clear(nTimeStamp:=0, bResetConfirmation:= FALSE);
		END_IF
	END_IF		
	
	//Error - Nakrętki nie dojechały do czujnika nad butelka
	IF tonVibrator2AndNotbCapsSensor.Q THEN
		IF NOT arfbAlarm[3].bActive THEN
			arfbAlarm[3].Raise(nTimeStamp:=0);
		END_IF
	ELSE	
		IF  arfbAlarm[3].bActive AND bReset THEN
			arfbAlarm[3].Clear(nTimeStamp:=0, bResetConfirmation:= FALSE);
		END_IF
	END_IF		
	
	//Error - Brak nakrętek w zbiorniku
	IF tonNoCapsHopperSensor.Q THEN
		IF NOT arfbAlarm[4].bActive THEN
			arfbAlarm[4].Raise(nTimeStamp:=0);
		END_IF
	ELSE	
		IF  arfbAlarm[4].bActive AND bReset THEN
			arfbAlarm[4].Clear(nTimeStamp:=0, bResetConfirmation:= FALSE);
		END_IF
	END_IF			
ELSE
	bError	:=FALSE;
		IF  arfbAlarm[0].bActive THEN
			arfbAlarm[0].Clear(nTimeStamp:=0, bResetConfirmation:= FALSE);
		END_IF
		IF  arfbAlarm[1].bActive THEN
			arfbAlarm[1].Clear(nTimeStamp:=0, bResetConfirmation:= FALSE);
		END_IF
		IF  arfbAlarm[2].bActive THEN
			arfbAlarm[2].Clear(nTimeStamp:=0, bResetConfirmation:= FALSE);
		END_IF
		IF  arfbAlarm[3].bActive THEN
			arfbAlarm[3].Clear(nTimeStamp:=0, bResetConfirmation:= FALSE);
		END_IF
		IF  arfbAlarm[4].bActive THEN
			arfbAlarm[4].Clear(nTimeStamp:=0, bResetConfirmation:= FALSE);
		END_IF	
END_IF


//-----------------------------------------------------------------------
IF bError AND NOT bStateError THEN

	IF eLastState = eRunning THEN
		bCycleNotDone						:= TRUE;
	END_IF
	eState 									:= E_Station.eError;
END_IF

//------------------------------------------------------------------------
(*Wyświetlanie błedu na wyjściu*)
bError							:= FALSE;
FOR nAlarmNumerator := 0 TO 19 DO
	bError						:= bError OR arfbAlarm[nAlarmNumerator].bActive;
END_FOR

(*Wyświetlanie błedu na wyjściu*)
bError;

(*Przepisywanie nazwy stacji*)
sErrorStationName 							:= WSTRING_TO_STRING(sStationName);
END_ACTION

ACTION ACT_Homing:
//BAZOWANIE
eState:=E_Station.eHomingDone;
END_ACTION

ACTION ACT_Inverter:
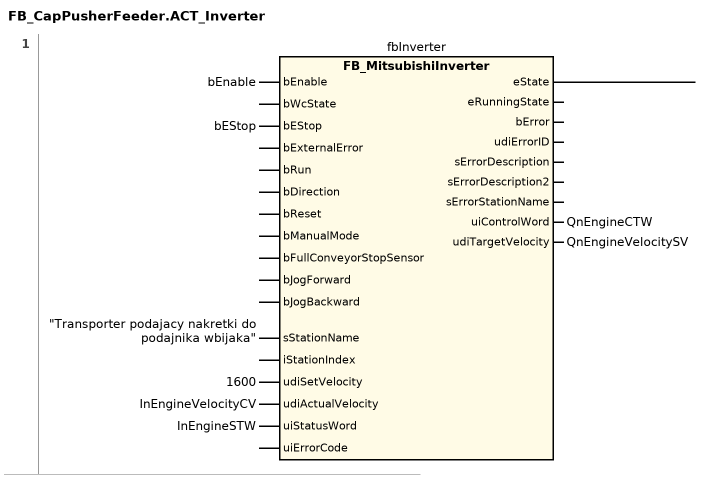
// NETWORK 1
fbInverter(
    bEnable := bEnable,
    bEStop := bEStop,
    sStationName := "Transporter podajacy nakretki do podajnika wbijaka",
    udiSetVelocity := 1600,
    udiActualVelocity := InEngineVelocityCV,
    uiStatusWord := InEngineSTW,
    uiControlWord => QnEngineCTW,
    udiTargetVelocity => QnEngineVelocitySV); // FB_MitsubishiInverter
END_ACTION

ACTION ACT_Limits:
IF iTimeToEmptySleeveError < 5 THEN
	iTimeToEmptySleeveError := 5;
END_IF
END_ACTION

ACTION ACT_ManualMovements:
//W trybie ruchów manualnych wykonuj ruchy za pomocą rozkazów manualnych
IF NOT bRun THEN
	fbInverter.bRun		:= bManualSorterEngine;
	bSorterVibrator		:= bManualSorterVibrator;
	bSorterVibrator2	:= bManualSorterVibrator2;	
	bSorterAir			:= bManualSorterAir;
END_IF

IF bHoming OR bHeightSet THEN
	eState:=E_Station.eHoming;
END_IF

IF bRun THEN	
	ACT_Running();
END_IF
//Zabezpieczenie przed kolizją stacji poprzez ruch podnośnika
END_ACTION

ACTION ACT_ResetCommands:
//Reset komend ruchu 	

fbInverter.bRun	:=	FALSE;
bSorterAir		:=	FALSE;
bSorterVibrator	:=	FALSE;
bSorterVibrator2:=	FALSE;
END_ACTION

ACTION ACT_Running:
//----------------------------------------------------------------------------------
// Obsługa podajnik zamknięc

CASE eRunningState OF
	
	//NIEGOTOWY
	E_CapFeederState.eDisabled:
		eRunningState			:=	E_CapFeederState.eReady;

	E_CapFeederState.eReady:
		fbInverter.bDirection 	:=	FALSE;
		IF bRun THEN
			iSortingCASE		:= 0;
			eRunningState		:=	E_CapFeederState.eSorting;
		END_IF
	
	E_CapFeederState.eSorting:
	
		// 	1-Najpierw powietrze
		//	2-Potem wibracje rekawa
		//	3-Potem wibracje kola jezeli nie ma na czujniku
		bSorterAir 				:= TRUE;			
		bSorterVibrator 		:= tonAirBeforeStart.Q;
		bSorterVibrator2 		:= TRUE;
		fbInverter.bRun 		:= fbbCapsWheelLevelSensor.bOut AND tonbSorterVibrator.Q ;
		
		CASE iSortingCASE OF 
			0:
				iSortingCASE			:=	iSortingCASE	+	10;
			
			10:
				fbInverter.bRun 		:= fbbCapsWheelLevelSensor.bOut AND tonbSorterVibrator.Q ;
				IF tonfbInverterbRun1.Q THEN //Chodzi 1s
					iSortingCASE		:=	iSortingCASE	+	10;
				END_IF
				
			20:
				fbInverter.bRun := FALSE;
				IF tonfbInverterbRun2.Q THEN //Stop 2s
					iSortingCASE	:=	10;
				END_IF
							
		END_CASE
			
		IF tonSortingEngineOff.Q THEN  //5S
			eRunningState 			:=E_CapFeederState.eSleeveFull;
		END_IF
	
	E_CapFeederState.eSleeveFull:
		bSorterVibrator 	:=	FALSE;		
		IF fbbCapsAndSleeveSensor.bOUT THEN
			bSorterVibrator2 	:= FALSE;
		ELSE
			bSorterVibrator2 	:= TRUE;
		END_IF
		fbInverter.bRun		:=	FALSE;
		bSorterAir			:=	NOT tonAirAfterStop.Q;
		IF tonAirAfterStop.Q THEN
			IF tonSortingEngineOn.Q THEN
				iSortingCASE		:= 0;
				eRunningState		:=E_CapFeederState.eSorting; 
			END_IF
		END_IF
	
	E_CapFeederState.eSleeveLowLevel:
	
		;
	
END_CASE
END_ACTION

ACTION ACT_Signals:
(** Timery na potrzeby bazowania**)
//Czujnik poziomu na kole
fbbCapsWheelLevelSensor		(bIN:=NOT bCapsWheelSensor AND eRunningState=E_CapFeederState.eSorting,		tFilterTimeOn:= T#8S, tFilterTimeOff:= T#40MS, bOUT=> );
fbbCapsWheelLevelSensor.bOut;

fbbCapsAndSleeveSensor		(bIN:=bCapsSleeveSensor AND bCapsSensor,		tFilterTimeOn:= T#2S, tFilterTimeOff:= T#100MS, bOUT=> );
tonbSorterVibrator			(IN:= bSorterVibrator, 					PT:=T#4S);
tonfbInverterbRun1			(IN:=fbInverter.bRun, 					PT:=T#600MS);
tonfbInverterbRun2			(IN:=NOT fbInverter.bRun, 				PT:=T#3S);


tonAirBeforeStart		(IN:=eRunningState=E_CapFeederState.eSorting, PT:=T#1S);
tonSortingEngineOff		(IN:=((eRunningState=E_CapFeederState.eSorting OR eRunningState=E_CapFeederState.eSleeveLowLevel) AND bRun AND bCapsSleeveSensor),PT:=INT_TO_TIME(iTimeDelayOff));
tonAirAfterStop			(IN:=eRunningState=E_CapFeederState.eSleeveFull, PT:=T#2S);
tonSortingEngineOn		(IN:=((eRunningState=E_CapFeederState.eSorting OR eRunningState=E_CapFeederState.eSleeveFull) AND bRun AND NOT bCapsSleeveSensor),PT:=INT_TO_TIME(iTimeDelayOn));
	
(** Timery używane podczas pracy stacji**)


(** Dodatkowy timer przy zatrzymywaniu**)
tonStoppingTime( IN:= eState= E_Station.eStopping, PT:=T#2S);
VIS_CP.IbCapPusher0DoorsOpen := NOT VIS_CP.IbCapPusher0DoorsOpen;
END_ACTION

ACTION ACT_Statistic:
//Statystyka do zliczania czasu cyklu 
rtrigCycleTimerRead(CLK:=eRunningState=E_CapFeederState.eSleeveFull OR eRunningState=E_CapFeederState.eSleeveLowLevel);

	IF rtrigCycleTimerRead.Q THEN
		tCycleTime:=tonCycleTimer.ET;
		
	END_IF
	
tonCycleTimer(IN:=eRunningState= E_CapFeederState.eSorting , PT:=T#1D);
END_ACTION

ACTION ACT_Status:

(*Zapisywanie ostatniego stanu*)
	IF eLastStateTemp<>eState THEN
		eLastState := eLastStateTemp;
	END_IF
	eLastStateTemp := eState;
	
	IF eLastRunningStateTemp<>eRunningState THEN
		eLastRunningState := eLastRunningStateTemp;
	END_IF
	eLastRunningStateTemp := eRunningState;
(*Koniec Zapisywanie ostatniego stanu*)
END_ACTION

ACTION ACT_Warnings:
//Usrawianie warningów

//Filtrowanie czujnika ultradźwiękowego
fbbLevelSensor	(bIN:=NOT bCapsSleeveSensor AND (eRunningState=E_CapFeederState.eSorting OR eRunningState=E_CapFeederState.eSleeveLowLevel OR eRunningState=E_CapFeederState.eSleeveFull) , tFilterTimeOn:= T#5S, tFilterTimeOff:=T#5S , bOUT=> );

IF fbbLevelSensor.bOUT THEN
		bWarning1						:=	TRUE;			
		udiWarningID					:=	1;
		sWarningDescription				:=	'Niski poziom w sorterze nasadek';
ELSE
		bWarning1						:=	FALSE;			
		udiWarningID					:=	0;
		sWarningDescription				:=	'';
END_IF
END_ACTION

ACTION aStationID:
udiStationID	:=	udiStationIndex;
END_ACTION

END_FUNCTION_BLOCK

// ---- POUs/FB/FB_CapPusher.TcPOU
(*
Nazwa:			FB_ROPPCapping
Opis:			
Wersja:			v0.1
Data:			2025-01-13
Autor:			DP
Urzadzenia:		
Konfiguracja:	
Info:
-
*)

FUNCTION_BLOCK FB_CapPusher
VAR_INPUT
	
	bEnable						: BOOL;					//Zezowlenie na pracę stacji sprawdzania
	bEStop						: BOOL;					//Stop Awaryjny nieaktywny
	bRun1						: BOOL;					//Włączenie 
	bHoming						: BOOL;					//Zezwolenie na wykonanie bazowania i pozycjonowania stacji sprawdzania
	bHeightSet					: BOOL;					//Bit do bazowania stacji na ustaloną wysokość 
	bIgnoreError				: BOOL;					//Ignorowania błędów cyklu pracy
	bReset						: BOOL;					//Reset błędu, jeśli w stanie "eError"
	iTime						: INT; 				
	iTime2						: INT; 				
	iTool						: INT;					//Wybór narzędzia (1-5), opisy w tablicy AsGripperScrewerTool	
	IbCapSensor					: BOOL;		
	IbPusherUpSensor			: BOOL;		
	IbPusherDownSensor			: BOOL;	
	IbBlockActuatorOnSensor		: BOOL;	
	IbBlockActuatorOffSensor	: BOOL;	
	IbFormPositioningUpSensor	: BOOL;		
	IbFormPositioningDownSensor : BOOL;	
	
	bManualMovement				: BOOL; 				//Uruchomienie trybu ruchów ręcznych
	udiStationIndex				: UDINT;				// Indywidualny numer stacji
	sStationName				: WSTRING;				// Nazwa stacji
	
END_VAR

VAR_OUTPUT
	eState						: E_Station;			// Aktualny stan stacju
	eRunningState				: E_GripperScrewer;		// Stan pracy stacji
	eRunningStateBeforeEstop	: E_GripperScrewer;  	// Stan przed Estope
	bError						: BOOL;					// Błąd stacji
	udiErrorID					: UDINT;				// Nr blędu przeciągania formatek
	sErrorDescription			: STRING(200);			// Opis błędu
	sErrorDescription2			: STRING(200);			// Opis błędu
	sErrorStationName			: STRING;				// Nazwa stacj
	udiStationID				: UDINT;				// Nr stacji

	bHomingNeeded				: BOOL;					// Wymagane ponowne bazowanie (blad podczas bazowania lub stop awaryjny)
	bHomingDone					: BOOL;					// Stacja zbazowana 
	bCycleDone1					: BOOL;					// Sygnał o zakończeniu cyklu
	bCycleNotDone1				: BOOL;					// Sygnał o niezakończonym cyklu	

	tCycleTime					: TIME;	 				// Czas cyklu 
	sWarningDescription			: STRING;
	bWarning1					: BOOL;
	udiWarningID				: UDINT;
	
	bCapPusher					: BOOL;
	bBlockActuator				: BOOL;
	bFormPositioning			: BOOL;
	
END_VAR

VAR_IN_OUT
	
	bManualCapPusher			: BOOL;
	bManualBlockActuator		: BOOL;
	bManualFormPositioning		: BOOL;

END_VAR

VAR

	// State
	eLastState					: E_Station;			//Stan ogólny bloku
	eLastStateTemp				: E_Station;			//Stan ogólny bloku
	eLastRunningState			: E_GripperScrewer;		//Stan podbloku
	eLastRunningStateTemp		: E_GripperScrewer;		//Stan podbloku

	bStateError					: BOOL;
	
	tonStoppingTime				: TON;					// Czasówka zbyt długiego zatrzymawania

	tonCycleTimer				: TON;					// Czasówka cyklu
	rtrigCycleTimerRead			: R_TRIG;				// Trigger do statystyk cyklu 
	rtResetCommands				: R_TRIG;

	tonCapPusherUp: TON;		
	tonBlockActuatorOn: TON;
	tonBlockActuatorOff: TON;	
	tonFormPositioningUp: TON;
	tonFormPositioningDown: TON;
		
	(*Ostrzeżenia*)

	(*Inne*)	
	fbCapSensor	:FB_InputFilter_v2;
	toneToPushing	:TON;
	toneHolding 	:TON;
	toneScrewing	:TON;
	toneGoingUp		:TON;
	
	//Zmienne od EVENTLOGGER
	bAlarmInit 						: BOOL := TRUE; 
	nAlarmNumerator					: INT;
	arfbAlarm						: ARRAY[0..19] OF  FB_TcAlarm;		//Tablica bloczków błędów
	fbSourceInfo 					: FB_TcSourceInfo;
	iSourceInfo						: I_TcSourceInfo;
	sAlarmTest						: STRING;
	//Koniec zmiennych od EVENTLOGGER
	
END_VAR

//Wywołanie bloczków od stacji. Ważna jest ich kolejność!!!
ACT_Limits();
ACT_ErrorHandling();
ACT_Signals();
ACT_Control();
ACT_Statistic();
ACT_Status();
ACT_Warnings();
aStationID();

ACTION ACT_Control:
	(*****Wyłączenie enable*****)
	IF NOT bEnable THEN
		IF eState <> E_Station.eDisabled AND eState <> E_Station.ePreparingToDisable THEN
				eState 				:= E_Station.ePreparingToDisable; 
		END_IF	
	END_IF

	(*****Estop*****)
	IF NOT bEstop  THEN	
		IF eState <> E_Station.eAborted AND eState <> E_Station.eAborting AND eState <> E_Station.eDisabled THEN
				eState 				:= E_Station.eAborting; 
		END_IF
	END_IF


	CASE eState OF
//--------------------------------------------------------------------------------
// Stan maszyny po wyłączeniu i przygotowanie do uruchomienia
	E_Station.eDisabled: 					// Stan nieaktywnosci (Stacja wyłączona) 
	
		IF bEnable THEN
			eState 				:= E_Station.ePreparingToReady; 
		END_IF 
		
//--------------------------------------------------------------------------------
// Stan maszyny po zatrzymaniu awaryjnym   
	E_Station.eAborted: 					// Stan bezpiecznego zatrzymania (po Abortingu) 

		IF bEStop THEN
			eState 				:= E_Station.ePreparingToReady;
		END_IF
		
//--------------------------------------------------------------------------------
// Stan maszyny naciśnieciu estopa 	
	E_Station.eAborting:                 	// Stan bezpiecznego zatrzymywania (po EStopie)

		ACT_ResetCommands();

		eState 						:=  E_Station.eAborted;  
		eRunningState				:=	E_GripperScrewer.eReady;
		
//--------------------------------------------------------------------------------
// Stan masyzny po wykryciu błędu			
	E_Station.eError:                 	 	// Stan błędu 	
		
		ACT_ResetCommands();
		
		IF bReset OR NOT bError THEN
			eState 					:= E_Station.eResetting;
			bError					:= FALSE;
		END_IF
		
//--------------------------------------------------------------------------------
// Stan masyzny po wykryciu błędu
	E_Station.eResetting:					// Stan resetowania bledu (po Errorze)
		
		IF NOT bError  THEN
			//{warning 'Sprawdzić błąd falownika CapFeeder'}
			udiErrorID 			:=	0;
			sErrorDescription 	:=	'';
			eState 				:=	E_Station.ePreparingToReady;
			eRunningState		:=	E_GripperScrewer.eReady;
		ELSE
			eState 				:=	E_Station.eError;
		END_IF
    
//--------------------------------------------------------------------------------
// Stan ruchoow manualnych
	E_Station.eManualMovement:     			// Stan ruchów manualnych  
   
		ACT_ManualMovements();
		//Wyjście z trybu serwisowego
		IF NOT bManualMovement THEN

			eState		:=	E_Station.eReady;
		END_IF
		
//--------------------------------------------------------------------------------
// Stan rozpoczecia bazowania
	E_Station.eHoming:						// Stan bazowania 
		
		ACT_Homing();
		IF NOT bHoming AND NOT bHeightSet THEN

		   eState							:=	E_Station.ePreparingToReady;
		END_IF		
		
//--------------------------------------------------------------------------------
// Stan zakończenia bazowania
	E_Station.eHomingDone:                  // Stan wykonania bazowania 
	

		bHomingDone							:=	TRUE;
		IF NOT bHoming AND NOT bHeightSet THEN
		   eState		:=	E_Station.eReady;
		END_IF
		
//--------------------------------------------------------------------------------
// Stan przygotowania do gotowości
	E_Station.ePreparingToReady:            // Stan przygotowywania do gotowosci (zawsze przed Ready)  

		eRunningState	:=	E_GripperScrewer.eReady;
		eState			:=	E_Station.eReady;	
		
//-------------------------------------------------------------------------------
// Stan przygotowania do wyłączenia maszyny
	E_Station.ePreparingToDisable:          // Stan przygotowywania do nieaktywnosci (po wyłączeniu Enable) 


		eRunningState			:=	E_GripperScrewer.eReady;		
		eState					:=	E_Station.eDisabled;

			
//--------------------------------------------------------------------------------
// Stan gotowości
	E_Station.eReady:						// Stan gotowosci 
	
		(*Skasowanie wszystkich komend*)
		IF rtResetCommands.Q THEN	ACT_ResetCommands();	END_IF
	
		IF bRun1  AND NOT bCycleDone1 AND NOT bCycleNotDone1 THEN
			eState 						:= E_Station.eStarting; 
		END_IF
		IF bHoming OR bHeightSet THEN
			eState 						:= E_Station.eHoming; 
		END_IF
		IF bManualMovement THEN
			bManualCapPusher			:=	bCapPusher;		
			bManualBlockActuator		:=	bBlockActuator;		
			bManualFormPositioning		:=	bFormPositioning;			
			eState 						:=	E_Station.eManualMovement; 
		END_IF
		IF NOT bRun1  THEN
			bCycleDone1 				:= FALSE;
			bCycleNotDone1 				:= FALSE;	
			bWarning1					:= FALSE;	
		END_IF
		
//--------------------------------------------------------------------------------
// Stan zatrzymywania
	E_Station.eStopping:					// Stan zatrzymywania 
		
		ACT_Running();

		IF tonStoppingTime.Q THEN
			ACT_ResetCommands();
			eRunningState							:= E_GripperScrewer.eReady;
			eState									:= E_Station.eReady;
		END_IF

		
//--------------------------------------------------------------------------------
// Stan uruchomienia lini ( po eReady)
	E_Station.eStarting:                  	// Stan uruchamiania (po Ready)

		eState					 := E_Station.eRunning; 

//--------------------------------------------------------------------------------
// Stan wykonywania pracy
	E_Station.eRunning:               		// Stan wykonywania cyklu (po Startingu), w tym stanie osobny

		ACT_Running();
		IF NOT bRun1 THEN					(*Przerywanie cyklu*)
			eState 				 := E_Station.eStopping;	
		END_IF
		IF (bCycleDone1 OR bCycleNotDone1)  THEN (*Cykl zakończony*)
			eState 				 := E_Station.eReady;
		END_IF						
		
		
END_CASE
END_ACTION

ACTION ACT_ErrorHandling:
// Alarm_0590	590	Error	Błąd górnej pozycji wbijaka - sprawdź czujnik lub odblokuj mechanicznie
// Alarm_0591	591	Error	Błąd wysunięcia siłownika bocznego - sprawdź wyłącznik
// Alarm_0592	592	Error	Błąd schowania siłownika bocznego - sprawdź czujnik lub odblokuj mechanicznie
// Alarm_0593	593	Error	Błąd wysunięcia siłownika podnoszenia formatki - sprawdź czujnik lub odblokuj mechanicznie
// Alarm_0594	594	Error	Błąd schowania siłownika podnoszenia formatki - sprawdź czujnik lub odblokuj mechanicznie

IF bAlarmInit THEN
    bAlarmInit := FALSE; 
	fbSourceInfo.Clear();
	fbSourceInfo.sName:=wsLiteral_TO_UTF8(sStationName);//'Machine';
	fbSourceInfo.nId:=udiStationID;//2700;
	// Alarm_0590	590	Error	Błąd górnej pozycji wbijaka - sprawdź czujnik lub odblokuj mechanicznie
    arfbAlarm[0].CreateEx(stEventEntry := TC_EVENTS.AlarmClass.Alarm_0590, bWithConfirmation:= FALSE,  ipSourceInfo:= fbSourceInfo); 
	// Alarm_0591	591	Error	Błąd wysunięcia siłownika bocznego - sprawdź wyłącznik
	arfbAlarm[1].CreateEx(stEventEntry := TC_EVENTS.AlarmClass.Alarm_0591, bWithConfirmation:= FALSE,  ipSourceInfo:= fbSourceInfo);
	// Alarm_0592	592	Error	Błąd schowania siłownika bocznego - sprawdź czujnik lub odblokuj mechanicznie
	arfbAlarm[2].CreateEx(stEventEntry := TC_EVENTS.AlarmClass.Alarm_0592, bWithConfirmation:= FALSE,  ipSourceInfo:= fbSourceInfo);
	// Alarm_0593	593	Error	Błąd wysunięcia siłownika podnoszenia formatki - sprawdź czujnik lub odblokuj mechanicznie
	arfbAlarm[3].CreateEx(stEventEntry := TC_EVENTS.AlarmClass.Alarm_0593, bWithConfirmation:= FALSE,  ipSourceInfo:= fbSourceInfo);
	// Alarm_0594	594	Error	Błąd schowania siłownika podnoszenia formatki - sprawdź czujnik lub odblokuj mechanicznie
	arfbAlarm[4].CreateEx(stEventEntry := TC_EVENTS.AlarmClass.Alarm_0594, bWithConfirmation:= FALSE,  ipSourceInfo:= fbSourceInfo);
END_IF

//OBSŁUGA BŁĘDÓW STACJI SPRAWDZANIA
//************LISTA BŁĘDÓW***************
bStateError:= (eState=E_Station.eError) OR (eState=E_Station.eResetting);
//************LISTA BŁĘDÓW***************

//Error 1 - podnośnik nie porusza się pomimo wysterowania 

IF (bEnable OR (eState = E_Station.ePreparingToDisable))  THEN
	
	tonCapPusherUp			(IN:= bEstop AND NOT bCapPusher AND NOT IbPusherUpSensor, 							PT:=T#300MS);
	tonBlockActuatorOn		(IN:= bEstop AND bBlockActuator AND NOT IbBlockActuatorOnSensor,					PT:=T#1S500MS);
	tonBlockActuatorOff		(IN:= bEstop AND NOT bBlockActuator AND NOT IbBlockActuatorOffSensor,				PT:=T#300MS);	
	//tonFormPositioningUp	(IN:= bEstop AND bFormPositioning AND NOT IbFormPositioningUpSensor,				PT:=T#300MS); //Czujnik górny zle widzi
	tonFormPositioningDown	(IN:= bEstop AND NOT bFormPositioning AND NOT IbFormPositioningDownSensor,			PT:=T#300MS);	
		
	//Error 
	IF tonCapPusherUp.Q THEN
		IF NOT arfbAlarm[0].bActive THEN
			arfbAlarm[0].Raise(nTimeStamp:=0);
		END_IF
	ELSE	
		IF  arfbAlarm[0].bActive AND bReset THEN
			arfbAlarm[0].Clear(nTimeStamp:=0, bResetConfirmation:= FALSE);
		END_IF
	END_IF		
	//Error 
	IF tonBlockActuatorOn.Q THEN
		IF NOT arfbAlarm[1].bActive THEN
			arfbAlarm[1].Raise(nTimeStamp:=0);
		END_IF
	ELSE	
		IF  arfbAlarm[1].bActive AND bReset THEN
			arfbAlarm[1].Clear(nTimeStamp:=0, bResetConfirmation:= FALSE);
		END_IF
	END_IF				
	//Error 
	IF tonBlockActuatorOff.Q THEN
		IF NOT arfbAlarm[2].bActive THEN
			arfbAlarm[2].Raise(nTimeStamp:=0);
		END_IF
	ELSE	
		IF  arfbAlarm[2].bActive AND bReset THEN
			arfbAlarm[2].Clear(nTimeStamp:=0, bResetConfirmation:= FALSE);
		END_IF
	END_IF		
	//Error 
	IF tonFormPositioningUp.Q THEN
		IF NOT arfbAlarm[3].bActive THEN
			arfbAlarm[3].Raise(nTimeStamp:=0);
		END_IF
	ELSE	
		IF  arfbAlarm[3].bActive AND bReset THEN
			arfbAlarm[3].Clear(nTimeStamp:=0, bResetConfirmation:= FALSE);
		END_IF
	END_IF	
	//Error 
	IF tonFormPositioningDown.Q THEN
		IF NOT arfbAlarm[4].bActive THEN
			arfbAlarm[4].Raise(nTimeStamp:=0);
		END_IF
	ELSE	
		IF  arfbAlarm[4].bActive AND bReset THEN
			arfbAlarm[4].Clear(nTimeStamp:=0, bResetConfirmation:= FALSE);
		END_IF
	END_IF	
	
ELSE
	bError	:=FALSE;
		bError	:=FALSE;
		IF  arfbAlarm[0].bActive THEN
			arfbAlarm[0].Clear(nTimeStamp:=0, bResetConfirmation:= FALSE);
		END_IF
		IF  arfbAlarm[1].bActive THEN
			arfbAlarm[1].Clear(nTimeStamp:=0, bResetConfirmation:= FALSE);
		END_IF
		IF  arfbAlarm[2].bActive THEN
			arfbAlarm[2].Clear(nTimeStamp:=0, bResetConfirmation:= FALSE);
		END_IF
		IF  arfbAlarm[3].bActive THEN
			arfbAlarm[3].Clear(nTimeStamp:=0, bResetConfirmation:= FALSE);
		END_IF
		IF  arfbAlarm[4].bActive THEN
			arfbAlarm[4].Clear(nTimeStamp:=0, bResetConfirmation:= FALSE);
		END_IF		
END_IF


//-----------------------------------------------------------------------
IF bError AND NOT bStateError THEN

	IF eLastState = eRunning THEN
		bCycleNotDone1						:= TRUE;
	END_IF

	eState 									:= E_Station.eError;
END_IF


//------------------------------------------------------------------------
(*Wyświetlanie błedu na wyjściu*)
bError							:= FALSE;
FOR nAlarmNumerator := 0 TO 19 DO
	bError						:= bError OR arfbAlarm[nAlarmNumerator].bActive;
END_FOR

(*Wyświetlanie błedu na wyjściu*)
bError;

(*Przepisywanie nazwy stacji*)
sErrorStationName 							:= WSTRING_TO_STRING(sStationName);

//Jezeli nie zbazowane to potrzebne bazowanie
END_ACTION

ACTION ACT_Homing:
//BAZOWANIE


eState:=E_Station.eHomingDone;
END_ACTION

ACTION ACT_Limits:

END_ACTION

ACTION ACT_ManualMovements:
//W trybie ruchów manualnych wykonuj ruchy za pomocą rozkazów manualnych
IF NOT bRun1  THEN			
	bCapPusher				:=	bManualCapPusher;		
	bBlockActuator			:=	bManualBlockActuator;		
	bFormPositioning		:=	bManualFormPositioning;				
ELSE	//Kasuje zeby po cyklu nic sie nie poruszało
	bManualCapPusher		:= FALSE;	
	bManualBlockActuator	:= FALSE;	
	bManualFormPositioning	:= FALSE;	
END_IF

IF bHoming OR bHeightSet THEN
	eState:=E_Station.eHoming;
END_IF

IF bRun1  THEN	
	ACT_Running();
END_IF

IF NOT bRun1  THEN
	bCycleDone1 				:= FALSE;
	bCycleNotDone1 				:= FALSE;	
	bWarning1					:= FALSE;	
END_IF

//Zabezpieczenie przed kolizją stacji poprzez ruch podnośnika
END_ACTION

ACTION ACT_ResetCommands:
//Reset komend ruchu 	

bCapPusher			:=	FALSE;
bBlockActuator		:=	FALSE;
bFormPositioning	:=	FALSE;
END_ACTION

ACTION ACT_Running:

CASE eRunningState OF

//====================================
	
	(*Oczekiwanie na wykonanie pojedynczego cyklu*)
	E_GripperScrewer.eReady:
	 		                                       	
		IF NOT bCycleDone1 AND NOT bCycleNotDone1  THEN                                           	
			IF bRun1 THEN                			
					eRunningState			:=	E_GripperScrewer.eToPushingPosition;	
			END_IF
		END_IF
		
//====================================		
	(*Ruch na pozycję *)			
	E_GripperScrewer.eToPushingPosition:
	
		bFormPositioning					:= TRUE;
		
		IF toneToPushing.Q THEN
			bBlockActuator					:= bRun1;	 
			IF fbCapSensor.bOUT THEN
				eRunningState					:=	E_GripperScrewer.eScrewing;	
			END_IF	
		END_IF

//====================================		
		
	(*Zakręcanie*)
	E_GripperScrewer.eScrewing:
		IF toneScrewing.Q THEN
			bCapPusher							:= bRun1;
			//IF IbPusherDownSensor THEN
				eRunningState					:=	E_GripperScrewer.eHolding;
			//END_IF
		END_IF
	
//====================================

	(*Przytrzymanie / Czas na odbpuszczenie chwytakow*)					
	E_GripperScrewer.eHolding:
	
		IF toneHolding.Q 		 THEN 
			eRunningState					:=	E_GripperScrewer.eGoingUp;			
		END_IF	

//====================================	

	(*Podnoszenie do góry / reset laga i obrót do pozycji gotowości*)			 
	E_GripperScrewer.eGoingUp:
	
		bCapPusher							:=	FALSE;
		bBlockActuator						:=	FALSE;	
		bFormPositioning					:=	FALSE;			
		IF toneGoingUp.Q THEN
			eRunningState 						:=	E_GripperScrewer.eDone;
		END_IF

		
//====================================			
	(*Zakręcono*)			
	E_GripperScrewer.eDone:
	
		bCycleDone1 						:=	bRun1;
		bCycleNotDone1						:=	NOT bRun1;
		eRunningState 						:=	E_GripperScrewer.eReady;					

//====================================	
			
	E_GripperScrewer.eNotDone:

		bCycleNotDone1 						:=	TRUE;
		eRunningState						:=	E_GripperScrewer.eReady;	
	
END_CASE
END_ACTION

ACTION ACT_Signals:
(** Timery na potrzeby bazowania**)
rtResetCommands			(CLK:=	eState = E_Station.eReady (* OR *)		,Q=>); //Triger do resetu zmienych

(** Timery używane podczas pracy stacji**)
fbCapSensor			(bIN:=	IbCapSensor OR bIgnoreError,									tFilterTimeOn:= T#60MS, tFilterTimeOff:= T#30MS, bOUT=> );
toneToPushing		(IN:=	eRunningState=E_GripperScrewer.eToPushingPosition,				PT:= T#50MS);
toneHolding			(IN:=	eRunningState=E_GripperScrewer.eHolding, PT:= INT_TO_TIME(iTime));
toneScrewing		(IN:=	eRunningState=E_GripperScrewer.eScrewing,							PT:= T#100MS);	
toneGoingUp			(IN:=	eRunningState=E_GripperScrewer.eGoingUp,						PT:= T#150MS);	

(** Dodatkowy timer przy zatrzymywaniu**)
tonStoppingTime( IN:= eState= E_Station.eStopping, PT:=T#2S);
END_ACTION

ACTION ACT_Statistic:
//Statystyka do zliczania czasu cyklu 
rtrigCycleTimerRead(CLK:=eRunningState=E_GripperScrewer.eDone );

	IF rtrigCycleTimerRead.Q THEN
		tCycleTime:=tonCycleTimer.ET;
	END_IF
	
	tonCycleTimer(IN:=eRunningState>E_GripperScrewer.eReady,PT:=T#1D);
END_ACTION

ACTION ACT_Status:

(*Zapisywanie ostatniego stanu*)
	IF eLastStateTemp<>eState THEN
		eLastState := eLastStateTemp;
	END_IF
	eLastStateTemp := eState;
	
	IF eLastRunningStateTemp<>eRunningState THEN
		eLastRunningState := eLastRunningStateTemp;
	END_IF
	eLastRunningStateTemp := eRunningState;
(*Koniec Zapisywanie ostatniego stanu*)
END_ACTION

ACTION ACT_Warnings:

END_ACTION

ACTION aStationID:
udiStationID	:=	udiStationIndex;
END_ACTION

END_FUNCTION_BLOCK

// ---- POUs/P00_Alarms.TcPOU
(*
Nazwa:			P00_Alarms
Opis:			Obsługa alarmów
Wersja:			v0.1
Data:			2018-10-10
Autor:			TW,DP
Urzadzenia:		Obsługa alarmów
Konfiguracja:	
Info:
- 80%
- dodać ewentualnie nowe alarmy w general alarms
#######################################################
#######################################################
*)
PROGRAM P00_Alarms

VAR CONSTANT
	STATION_COUNT														: INT :=90;
END_VAR

VAR
	aLastStationsErrors													: ARRAY [1..STATION_COUNT] OF S_Error;
	aStationsErrors														: ARRAY [1..STATION_COUNT] OF S_Error;
	
	i																	: INT;
	nCountSaveLastError													: INT;
	nCountertooLong														: INT;
	iWarningAcknowledgeAll												: INT;
	iCounterFormsAfterScrewer											: INT;
	
	// Wyłaczenie resetu po 2 s
	tonResetOff															: TON;
	tonFuseFB1OK														: TON;	
	tonFuseFB2OK														: TON;
	tonDCSupply1OK														: TON;	
	tonDCSupply2OK														: TON;	
	tonDCSupply3OK														: TON;	
	tonSoftAlarm														: TON;
	tonFirstCycle														: TON;	
	tonSystemDiagnosisError												: TON;
	tonPowerSuppyTerminal1UsUndervoltageError							: TON;
	tonPowerSuppyTerminal2UpUndervoltageError							: TON;
	tonPowerSuppyTerminal2UsUndervoltageError							: TON;
	tonBottleCheckAfterBottleTransferSensor								: TON;
	tonIbBottleNotInserted												: TON;
	tonResetFuseBlock													: TON;
	TimerWatchdog_eUndefined											: TON;
	TimerWatchdog_eAborting												: TON;
	TimerWatchdog_eResetting											: TON;
	TimerWatchdog_eStopping												: TON;
	TimerWatchdog_eIdleAndNotStationsAreReady							: TON;
	tonFormsStuckAfterScrewersAlarm										: TON;
	tonFormsStuckAfterLidSealerAlarm									: TON;
	tonFormsStuckAfterROPPAlarm											: TON;
	tonFormsStuckAfterCapSorterAlarm									: TON;
	rtWarningOccure0													: R_TRIG;
	rtWarningOccure1													: R_TRIG;
	rtWarningOccure2													: R_TRIG;
	rtWarningOccure4													: R_TRIG;              													
	rtWarningOccure3													: R_TRIG;
	rtWarningOccure5													: R_TRIG;
	rtWarningOccure6													: R_TRIG;	
	rtWarningOccure7													: R_TRIG;	
	rtWarningOccure8													: R_TRIG;
	rtWarningOccure9													: R_TRIG;
	rtWarningOccure10													: R_TRIG;
	rtWarningOccure11													: R_TRIG;
	rtWarningOccure12													: R_TRIG;
	rtWarningOccure13													: R_TRIG;
	rtWarningOccure14													: R_TRIG;
	rtWarningOccure15													: R_TRIG;
	rtWarningOccure16													: R_TRIG;
	rtWarningOccure17													: R_TRIG;
	rtWarningOccure18													: R_TRIG;
	rtWarningOccure19													: R_TRIG;
	rtWarningOccure20													: R_TRIG;
	rtWarningOccure21													: R_TRIG;
	rtWarningOccure22													: R_TRIG;
	rtEmergencyStop														: R_TRIG;
	rtMachineStateAborting												: R_TRIG;

	tonCompressedAir: TON;
	rtWarningOccure23: R_TRIG;
	rtWarningOccure24: R_TRIG;
	rtWarningOccure25: R_TRIG;
	rtWarningOccure26: R_TRIG;	
	rtWarningOccure27: R_TRIG;		
	rtWarningOccure28: R_TRIG;		
	rtWarningOccure29: R_TRIG;		
	rtWarningOccure30: R_TRIG;		
	rtWarningOccure31: R_TRIG;		
	rtWarningOccure32: R_TRIG;		
	rtWarningOccure33: R_TRIG;		
	rtWarningOccure34: R_TRIG;		
	rtWarningOccure35: R_TRIG;	
	rtWarningOccure36: R_TRIG;	
	rtWarningOccure37: R_TRIG;
	rtWarningOccure38: R_TRIG;
	rtWarningOccure39: R_TRIG;
	rtWarningOccure40: R_TRIG;
	rtWarningOccure41: R_TRIG;
	rtWarningOccure42: R_TRIG;
	
	tonBadBottleConvoyerAlarm: TON;
	tonFormStuckBeforeDispencer14Alarm: TON;	
	tonFormStuckAfterDispencer34Alarm: TON;
	tonbFormsStuckBeforeScrewersAlarm: TON;
	tonFormsStuckBeforeScrewersAlarm2: TON;
	tonFormsStuckBeforeScrewersAlarm3: TON;
	tonFormsStuckBeforeCapSorterAlarm: TON;
	tonFormStuckAfterDispencerAlarm: TON;
	tonstBottleSorterReadiWatchdog: TON;
	tonstCapSorterReadiWatchdog: TON;	
	(*Bład sortera nasadek*)
	rtiCapFeederCheckCountNOK	: R_TRIG;
	(*Bład komunikacji*)
	iBottleSorterReadLastWatchdog		: INT;
	iCapSorterReadLastWatchdog			: INT;
	(*Inny*)
	
	bWarningTest: BOOL;
	j: INT;
	tonActiveWarning: TON;
	uliWarningAcknowledgeTemp: ULINT;
	rtWarningNew: R_TRIG;
	tonWarningNew: TON;
	tonbFormsDragingRightRunCheck: TON;
	tonbFormsDragingLeftRunCheck: TON;	
	AudiActiveWarningDescriptionIDtemp						:ARRAY [0..63] OF UDINT;	// ID warningów do tłumaczeń na wizualizacji
tonEmergencyStop:TON;

	//Zmienne od EVENTLOGGER
	bAlarmInit 						: BOOL := TRUE; 
	nAlarmNumerator					: INT;
	arfbAlarm						: ARRAY[0..79] OF  FB_TcAlarm;		//Tablica bloczków błędów
	fbSourceInfo 					: FB_TcSourceInfo;
	iSourceInfo						: I_TcSourceInfo;
	sAlarmTest						: STRING;
	hrOccuredErrorCode  			: HRESULT;
    hrOccuredErrorCodeHistory  		: HRESULT;
	//Koniec zmiennych od EVENTLOGGER	


END_VAR

rtMachineStateAborting(CLK := P00_PackML.fbPMLAuto.ePMLState = E_PMLState.ePMLState_ABORTING, Q =>);

aAlarms();
aGeneralAlarms();
aWarnings();
aCommunicationError();
aActiveWarnings();

//OBSŁUGA BŁĘDÓW I WYSYŁANIE ICH DO WIZUALIZACJI

